METHOD M_GetAllProps : ERRORID
VAR_INPUT
	refCmdData : REFERENCE TO  ST_CmdData;
END_VAR
SUPER^.M_GetAllProps(refCmdData);
nCurrentPropIndex := nCurrentPropIndex + 1;
refCmdData.n32Data[nCurrentPropIndex] := REAL_TO_DINT(rWorkingDistance);
nCurrentPropIndex := nCurrentPropIndex + 1;
refCmdData.n32Data[nCurrentPropIndex] := BOOL_TO_DINT(bInvertWorkingDistance);
nCurrentPropIndex := nCurrentPropIndex + 1;
refCmdData.n32Data[nCurrentPropIndex] := eLightOutput;
nCurrentPropIndex := nCurrentPropIndex + 1;
refCmdData.n32Data[nCurrentPropIndex] := nLightOutputChannel;
END_METHOD

METHOD M_SetAllProps : ERRORID
VAR_INPUT
	refCmdData : REFERENCE TO  ST_CmdData;
END_VAR
M_SetAllProps := SUPER^.M_SetAllProps(refCmdData);

IF M_SetAllProps > 0 THEN
	RETURN;
END_IF

//WorkingDistance
nCurrentPropIndex := nCurrentPropIndex + 1;
nSpecPropIndex := nCurrentPropIndex;
rWorkingDistance := DINT_TO_REAL(refCmdData.n32Data[nCurrentPropIndex]);
nCurrentPropIndex := nCurrentPropIndex + 1;
bInvertWorkingDistance := DINT_TO_BOOL(refCmdData.n32Data[nCurrentPropIndex]);

//LightOutput
nCurrentPropIndex := nCurrentPropIndex + 1;
eLightOutput := DINT_TO_USINT(refCmdData.n32Data[nCurrentPropIndex]);

//LightOutputChannel
nCurrentPropIndex := nCurrentPropIndex + 1;
nLightOutputChannel := DINT_TO_USINT(refCmdData.n32Data[nCurrentPropIndex]);

nNoOfProps := nCurrentPropIndex + 1;
END_METHOD

METHOD M_SetSingleProp : ERRORID
VAR_INPUT
	refCmdData : REFERENCE TO  ST_CmdData;
END_VAR
IF nSpecPropIndex = refCmdData.aHeader[1] THEN
	rWorkingDistance := DINT_TO_REAL(refCmdData.n32Data[0]);
ELSIF nSpecPropIndex + 1 = refCmdData.aHeader[1] THEN
	bInvertWorkingDistance := DINT_TO_BOOL(refCmdData.n32Data[0]);
ELSIF nSpecPropIndex + 3 = refCmdData.aHeader[1] THEN
	nLightOutputChannel := DINT_TO_USINT(refCmdData.n32Data[0]);
ELSE
	M_SetSingleProp := SUPER^.M_SetSingleProp(refCmdData);
END_IF
END_METHOD

PROPERTY P_stAbsPosTotal : ST_3DPoint
GET
VAR
	stPosTemp : ST_3DPoint;
END_VAR
stPosTemp := SUPER^.P_stAbsPosPhys;
IF bInvertWorkingDistance THEN
	stPosTemp.Z := stPosTemp.Z + rWorkingDistance;
ELSE
	stPosTemp.Z := stPosTemp.Z - rWorkingDistance;
END_IF
P_stAbsPosTotal := stPosTemp;
END_GET
END_PROPERTY

PROPERTY P_stCurrentPosTotal : ST_3DPoint
GET
VAR
	stPosTemp : ST_3DPoint;
END_VAR
stPosTemp := P_stCurrentPosPhys;
IF bInvertWorkingDistance THEN
	stPosTemp.Z := stPosTemp.Z + rWorkingDistance;
ELSE
	stPosTemp.Z := stPosTemp.Z - rWorkingDistance;
END_IF
P_stCurrentPosTotal := stPosTemp;
END_GET
END_PROPERTY

END_FUNCTION_BLOCK

// ---- Objects/Tools/FB_ZLevelSensor.TcPOU
FUNCTION_BLOCK FB_ZLevelSensor EXTENDS FB_MzTool
VAR_INPUT
END_VAR
VAR_OUTPUT
END_VAR
VAR
	rCurrentZMeasPos	: REAL;
	rZMeasPosOffset		: REAL;
END_VAR

SUPER^();	//FB_MzTool aufrufen

//Prozessdaten aktualisieren
IF pZAxisRef > 0 THEN
	stProcessData.n32Data[7] := BOOL_TO_DINT(pZAxisRef^.stInput.nToolState.1);
END_IF
aObjProcData[nNotifyId] := stProcessData;

ACTION A_Reset:
nStateA_ResetSpec := 80;
SUPER^.A_Reset();
END_ACTION

METHOD FB_init : BOOL
VAR_INPUT
	bInitRetains : BOOL; // if TRUE, the retain variables are initialized (warm start / cold start)
	bInCopyCode : BOOL;  // if TRUE, the instance afterwards gets moved into the copy code (online change)
END_VAR
eObjectType := E_ObjectType.OBJECTTYPE_ZSensor;
eObjectGroup := E_ObjectGroup.OBJECTGROUP_MzTool OR E_ObjectGroup.OBJECTGROUP_Device;
END_METHOD

METHOD M_AddChild : ERRORID
VAR_INPUT
	pObject : POINTER TO FB_Object;
	nSlotNr	: UINT;
	nIndex 	: INT;
END_VAR
//Kann keine Objekte aufnehmen
M_AddChild := E_ErrorIdObjMgmt.ERRORID_ObjectCanNotTakeChilds;
END_METHOD

METHOD M_CheckAction : ERRORID
VAR_INPUT
	refActionData 	: REFERENCE TO ST_ActionData;
	pCorrelObject	: POINTER TO FB_Object;
END_VAR

VAR
	eMeasureMode : E_MeasureMode;
	pInkStation	 : POINTER TO FB_InkStation;
END_VAR
CASE refActionData.eAction OF
	E_Action.ACTION_MeasureTool:
		//ZSensor montiert?
		IF NOT P_bSensorMounted THEN
			M_CheckAction := E_ErrorIdCmd.ERRORID_ZSensorNotMounted;
		END_IF
		//MeasureMode auswerten
		eMeasureMode := DINT_TO_USINT(refActionData.aParams[1]);
		IF eMeasureMode = E_MeasureMode.MEAS_MODE_Auto THEN	//Target muss passend sein
			CASE fbObjectDirectory.M_GetObjType(refActionData.nTarget) OF
				E_ObjectType.OBJECTTYPE_InkStation:
					pInkStation := fbObjectDirectory.M_GetObjPointer(refActionData.nTarget);
					//Inkstation offen?
					IF (pInkStation^.P_eCoverState <> E_OpClState.Open) THEN
						M_CheckAction := E_ErrorIdCmd.ERRORID_InkStationNotOpen;
						RETURN;
					END_IF
					//Inkstation im Stillstand?
					IF(pInkStation^.P_nCurrentSpinSpeed <> 0) THEN
						M_CheckAction := E_ErrorIdCmd.ERRORID_InkStationIsStillSpinning;
						RETURN;
					END_IF
				E_ObjectType.OBJECTTYPE_DryPad,
				E_ObjectType.OBJECTTYPE_Slide,
				//E_ObjectType.OBJECTTYPE_Wafer,
				E_ObjectType.OBJECTTYPE_Point:
				//Do nothing
			ELSE
				M_CheckAction := E_ErrorIdCmd.ERRORID_UnsuitableTarget;
				RETURN;
			END_CASE
		
		ELSIF eMeasureMode = E_MeasureMode.MEAS_MODE_SemiAuto THEN	//Target muss erst ermittelt werden
			//nMeasToolTargetIdx := aI_MzTool[nMeasToolMzToolIdx].M_GetCurrentTargetIdx();
			//passendes Target gefunden?
			(*IF NOT (aI_Target[nMeasToolTargetIdx].P_eObjectType = E_ObjectType.OBJECTTYPE_Slide OR 
				aI_Target[nMeasToolTargetIdx].P_eObjectType = E_ObjectType.OBJECTTYPE_DryPad OR
				aI_Target[nMeasToolTargetIdx].P_eObjectType = E_ObjectType.OBJECTTYPE_Wafer) THEN
				M_ExeAction := E_ErrorIdCmd.ERRORID_InvalidTarget;
				RETURN;					
			END_IF*)
			;
		ELSE
			M_CheckAction := E_ErrorIdCmd.ERRORID_InvalidMeasureMode;
			RETURN;
		END_IF	
ELSE
	M_CheckAction := SUPER^.M_CheckAction(refActionData, pCorrelObject);	
END_CASE
END_METHOD

METHOD M_SetAllProps : ERRORID
VAR_INPUT
	refCmdData : REFERENCE TO  ST_CmdData;
END_VAR

VAR
	pExtruder : POINTER TO FB_Extruder;
END_VAR
IF pParentMzTool^.P_eObjectType = E_ObjectType.OBJECTTYPE_SinglePiezoHolder THEN
	;	
ELSIF pParentMzTool^.P_eObjectType = E_ObjectType.OBJECTTYPE_Extruder THEN
	pExtruder := pParentMzTool;
	IF pExtruder^.P_eExtruderType <> E_ExtruderType.SyringeExtruder1 THEN
		M_SetAllProps := E_ErrorIdObjMgmt.ERRORID_InvalidParentMzTool;
		RETURN;	
	END_IF
ELSE
	M_SetAllProps := E_ErrorIdObjMgmt.ERRORID_InvalidParentMzTool;
	RETURN;	
END_IF

M_SetAllProps := SUPER^.M_SetAllProps(refCmdData);
END_METHOD

PROPERTY P_bCollFree : BOOL
GET
VAR
	st3DPoint 		: ST_3DPoint;
END_VAR
//wenn Z-Stift nicht montiert, dann kollisionsfrei
IF pZAxisRef^.stInput.nToolState.1 THEN
	P_bCollFree := SUPER^.P_bCollFree;
ELSE
	P_bCollFree := TRUE;
END_IF
END_GET
END_PROPERTY

PROPERTY P_bSensorMounted : BOOL
GET
IF pParentMzTool^.P_eObjectType = E_ObjectType.OBJECTTYPE_SinglePiezoHolder OR pParentMzTool^.P_eObjectType = E_ObjectType.OBJECTTYPE_Extruder THEN
	P_bSensorMounted := pZAxisRef^.stInput.nToolState.1;	
END_IF
END_GET
END_PROPERTY

PROPERTY P_rToolRadius : REAL
GET
VAR
	stDim : ST_3DDimension;
END_VAR
P_rToolRadius := 1500.0;
END_GET
END_PROPERTY

END_FUNCTION_BLOCK

// ---- Objects/Targets/Active/FB_InkStation.TcPOU
FUNCTION_BLOCK FB_InkStation EXTENDS FB_ActiveTarget IMPLEMENTS I_TargetZSensor

VAR
	//Hardware-Verküpfung
	pSpinDrive			: POINTER TO FB_HwRefInkStatDriveSpin;
	pCoverDrive			: POINTER TO FB_HwRefInkStatDriveCover;
	//Hardware-Bausteine
	fbInitSpinDrive		: FB_InkStationInitSpinDrive;
	fbInitSpinCover		: FB_InkStationInitCoverDrive;
	fbOpenCloseCover	: FB_InkStationOpenClose;
	
	
	//Variablen allgemeine Statemachine
	eBasicAction		: E_Action;
	
	//Prozessdaten
	nCurrentSpinSpeed	: INT;
	bVacuumOn			: BOOL;
	
	//Spec-Properties
	nNoOfSpecPoints : USINT;
	stMeasurePoint		: ST_3DPoint;
	stInkPoint			: ST_3DPoint;
	nValveNrVac			: USINT;	//VentilNr Vakuum (FBox)
	nMinHoldVac			: INT;		//minimales Haltevakuum um zu Schleudern
	
	//****************************************Aktionvariablen****************************************************
	bActionLock			: ARRAY[50..150] OF BOOL;
	
	
	//Action: "Spin"
	bSpin				: BOOL;	
	nStateA_Spin		: USINT;			//State von A_Spin();
	
	timerSpin			: TON;				//Timer für Schleuderzeit
	tSpinTime			: TIME; 			//Schleuderzeit (bei 0 wird dauerhaft eingeschalten bis zum Ausschalten)
	nSpinSpeed			: INT;				//Drehzahl Schleuder RPM
	
	//Action: "OpenClose"
	bOpenClose			: BOOL;
	nStateA_OpenClose	: USINT;	//Statemachine von A_OpenClose();
	eOpClCtrl			: E_OpClCtrl;

END_VAR

{IF defined (variable:aFbInkStatDrvSpinRef)}
IF bInitFB THEN
	bInitFB := FALSE;
	F_CreateLinkedListHnd( ADR( aNodes ), SIZEOF( aNodes ), hList );
	//Fehlerstruktur vorausfüllen
	stError.ObjectId := nObjectID;
	stError.HardwareGrp := E_HardwareGrp.Nothing;
	stError.POU := E_POU.POU_FB_InkStation;
END_IF
IF (pSpinDrive = 0) OR  (pCoverDrive = 0) THEN
	RETURN;
END_IF

bIsInit := pSpinDrive^.bIsInit AND pCoverDrive^.bIsInit;
nCurrentSpinSpeed := pSpinDrive^.nCurrentSpeed  * 3;	//RPM

CASE eCurrentState OF
	E_MachineState.MACHINESTATE_Active:
		//BasicActions ausführen
		IF bInit THEN	//Initialisieren
			A_Init();
			IF nStateA_Init >= 80 THEN
				IF nStateA_Init >= 99 THEN
					bError := TRUE;	
				END_IF
				bInit := FALSE;
				nStateA_Init := 0;
				M_RemoveListEntry(nSearchValue:= E_Action.ACTION_Init);
			END_IF
		END_IF
		
		IF bSpin THEN	//Drehzahl Schleuder vorgeben
			A_Spin();
			IF nStateA_Spin >= 80 THEN
				IF nStateA_Spin >= 99 THEN
					bError := TRUE;	
				END_IF
				bSpin := FALSE;
				nStateA_Spin := 0;
				M_RemoveListEntry(nSearchValue:= E_Action.ACTION_InkSpin);
			END_IF
		END_IF		
		
		IF bOpenClose THEN	//Deckel auf/zu
			A_OpenClose();
			IF nStateA_OpenClose >= 80 THEN
				IF nStateA_OpenClose >= 99 THEN
					bError := TRUE;	
				END_IF
				bOpenClose := FALSE;
				nStateA_OpenClose := 0;
				M_RemoveListEntry(nSearchValue:= E_Action.ACTION_InkOpClCover);
			END_IF
		END_IF		
		
		IF bStop THEN
			A_Stop();
			IF nStateA_Stop >= 80 THEN
				IF nStateA_Stop >= 99 THEN
					bError := TRUE;
				END_IF
				M_RemoveListEntry(nSearchValue:= E_Action.ACTION_Stop);
				nStateA_Stop := 0;
				bStop := FALSE;
			END_IF							
		END_IF		
		
		IF hList.nCount = 0 THEN
			eCurrentState := E_MachineState.MACHINESTATE_Ready;
		END_IF

		IF bError  THEN
			eCurrentState := E_MachineState.MACHINESTATE_Error;
		END_IF

	E_MachineState.MACHINESTATE_Reset:
		A_Reset();
		IF nStateA_Reset = 80 THEN
			nStateA_Init := 0;
			nStateA_Spin := 0;
			nStateA_OpenClose := 0;
			nStateA_Stop := 0;
			nStateA_Reset := 0;
			bBusy := FALSE;
			bError := FALSE;
			bStopAllOnError := FALSE;
			fbList.A_Reset( hList := hList);
			MEMSET(ADR(bActionLock),0,SIZEOF(bActionLock));
			nErrorId := 0;
			stError.Cmd := 0;
			stError.ErrorId := 0;
			eCurrentState := E_MachineState.MACHINESTATE_Idle;
		ELSIF
			nStateA_Reset = 99 THEN
			fbErrorList.M_Add(stError);
			nStateA_Reset := 0;
			bBusy := FALSE;
			bError := TRUE;
			eCurrentState := E_MachineState.MACHINESTATE_Error;			
		END_IF
	
	E_MachineState.MACHINESTATE_Ready:
		bBusy := FALSE;
		eCurrentState := E_MachineState.MACHINESTATE_Idle;
	
	E_MachineState.MACHINESTATE_Error:
		pSpinDrive^.nSpeed := 0;
		bBusy := FALSE;
END_CASE

//Prozessdaten aktualisieren
stProcessData.nObjId := nObjectID;
stProcessData.n32Data[0] := BOOL_TO_DINT(bIsInit);
stProcessData.n32Data[1] := eCurrentState;
stProcessData.n32Data[2] := stError.ErrorId;
stProcessData.n32Data[3] := pSpinDrive^.nCurrentSpeed;
stProcessData.n32Data[4] := pCoverDrive^.P_eCoverState;
stProcessData.n32Data[5] := BOOL_TO_DINT(bVacuumOn);
stProcessData.n32Data[6] := pSpinDrive^.nCurrentVacuum;

aObjProcData[nNotifyId] := stProcessData;
{END_IF}

ACTION A_Init:
stError.POUState := nStateA_Init;

CASE nStateA_Init OF
	0:	//Spin initialisieren
		fbInitSpinDrive(pDriveRef:= pSpinDrive, bExecute:= TRUE);
		IF NOT fbInitSpinDrive.bBusy THEN
			IF fbInitSpinDrive.bError THEN
				stError.ErrorId := fbInitSpinDrive.nErrorId;
				nStateA_Init := 99;
			ELSE
				nStateA_Init := 1;			
			END_IF
			fbInitSpinDrive(bExecute:= FALSE);
		END_IF
	
	1: //Cover initialisieren
		fbInitSpinCover(pDriveRef:= pCoverDrive, bExecute:= TRUE);
		IF NOT fbInitSpinCover.bBusy THEN
			IF fbInitSpinCover.bError THEN
				stError.ErrorId := fbInitSpinCover.nErrorId;
				nStateA_Init := 99;
			ELSE
				nStateA_Init := 80;
			END_IF
			fbInitSpinCover(bExecute:= FALSE);
		END_IF
		
	70:	//Abbrechen
		nStateA_Init := 80;
		fbInitSpinDrive();
		IF fbInitSpinDrive.bBusy THEN
			nStateA_Init := 70;
			fbInitSpinDrive.M_Stop();
		ELSE
			fbInitSpinDrive(bExecute:= FALSE);
		END_IF
		fbInitSpinCover();
		IF fbInitSpinCover.bBusy THEN
			nStateA_Init := 70;
			fbInitSpinCover.M_Stop();
		ELSE
			fbInitSpinCover(bExecute:= FALSE);
		END_IF
END_CASE

//Errorhandling
IF nStateA_Init = 99 THEN
	stError.Cmd := E_Action.ACTION_Init;
	stError.POUAction := E_POUACT.POUACT_A_Init;
	fbErrorList.M_Add(stError);
END_IF
END_ACTION

ACTION A_OpenClose:
stError.POUState := nStateA_OpenClose;

IF nStateA_OpenClose = 0 THEN
	fbOpenCloseCover(pDriveRef:= pCoverDrive, eCtrl:= eOpClCtrl, bExecute:= TRUE); 
	IF NOT fbOpenCloseCover.bBusy THEN
		IF fbOpenCloseCover.bError THEN
			stError.ErrorId := fbOpenCloseCover.nErrorId;
			nStateA_OpenClose := 99;
		ELSE
			nStateA_OpenClose := 80;
		END_IF
		fbOpenCloseCover(bExecute:= FALSE); 
	END_IF
END_IF

//Errorhandling
IF nStateA_OpenClose = 99 THEN
	stError.Cmd := E_Action.ACTION_InkOpClCover;
	stError.POUAction := E_POUACT.POUACT_A_OpenClose;
	fbErrorList.M_Add(stError);
END_IF
END_ACTION

ACTION A_Reset:
CASE nStateA_Reset OF
	0:
		nStateA_Reset := 80;
END_CASE
END_ACTION

ACTION A_Spin:
IF pSpinDrive^.nStatus.3 THEN	//Error
	stError.POUState := nStateA_Spin;
	nStateA_Spin := 99;
END_IF

CASE nStateA_Spin OF
	0:
		pSpinDrive^.nSpeed := nSpinSpeed;
		IF tSpinTime > T#0S THEN
			timerSpin(IN:= TRUE, PT:= tSpinTime);
		END_IF
		nStateA_Spin := 1;
		
	1:	//Überwachung Vacuum, Timer, Drezahl
		pSpinDrive^.nSpeed := nSpinSpeed;
		timerSpin();
		IF timerSpin.Q OR (pSpinDrive^.nSpeed = 0 AND pSpinDrive^.nCurrentSpeed = 0) OR nMinHoldVac < pSpinDrive^.nCurrentVacuum THEN
			timerSpin(IN:= FALSE);	
			pSpinDrive^.nSpeed := 0;
			nStateA_Spin := 2;
		END_IF
		
	2:	//Warten bis Drehzahl auf 0
		IF pSpinDrive^.nCurrentSpeed = 0 THEN
			nStateA_Spin := 80;
		END_IF
		
	70:	//Abbrechen
		timerSpin(IN:= FALSE);
		pSpinDrive^.nSpeed := 0;
		nStateA_Spin := 71;
		
	71:	//Speed = 0?
		IF pSpinDrive^.nCurrentSpeed = 0 THEN
			nStateA_Spin := 80;
		END_IF
		
END_CASE

//Errorhandling
IF nStateA_Spin = 99 THEN
	stError.Cmd := E_Action.ACTION_InkSpin;
	stError.POUAction := E_POUACT.POUACT_A_Spin;
	fbErrorList.M_Add(stError);
END_IF
END_ACTION

ACTION A_Stop:
CASE nStateA_Stop OF
	0:	
		IF bInit THEN
			nStateA_Init := 70;	
		END_IF
		
		IF bSpin THEN
			nStateA_Spin := 70;
		END_IF
		
		nStateA_Stop := 1;
	
	1:	//Warten bis alle Actions außer Stop abgebrochen sind
		IF hList.nCount = 1 THEN	//nur der Eintrag von Stop
			nStateA_Stop := 80;
		END_IF
END_CASE

//Errorhandling
IF nStateA_Stop = 99 THEN
	stError.Cmd := E_Action.ACTION_Stop;
	stError.POUAction := E_POUACT.POUACT_A_Stop;
	fbErrorList.M_Add(stError);
END_IF
END_ACTION

METHOD FB_init : BOOL
VAR_INPUT
	bInitRetains : BOOL; // if TRUE, the retain variables are initialized (warm start / cold start)
	bInCopyCode : BOOL;  // if TRUE, the instance afterwards gets moved into the copy code (online change)
END_VAR
eObjectType := E_ObjectType.OBJECTTYPE_InkStation;
eObjectGroup := E_ObjectGroup.OBJECTGROUP_Target OR E_ObjectGroup.OBJECTGROUP_Device;
END_METHOD

METHOD M_ApplyPos : ERRORID
VAR_INPUT
	eTargetRef 		: E_TargetRef;
	nPointSlotNr	: UINT;
	stPos 			: ST_3DPoint;
	bXPos			: BOOL;
	bYPos			: BOOL;
	bZPos			: BOOL;	
END_VAR
VAR
	stAbsPos		: ST_3DPoint;
END_VAR
IF eTargetRef = E_TargetRef.TARGETREF_SpecPoint THEN
	IF nPointSlotNr = 2 THEN
		stAbsPos := P_stAbsPosLB;
		IF bXPos THEN
			stInkPoint.X := stPos.X - stAbsPos.X;
		END_IF
		IF bYPos THEN
			stInkPoint.Y := stPos.Y - stAbsPos.Y;
		END_IF
		IF bZPos THEN
			stInkPoint.Z := stPos.Z - stAbsPos.Z;
		END_IF
	ELSE
		M_ApplyPos := E_ErrorIdCmd.ERRORID_InvalidTargetPointNr;
	END_IF
ELSE
	M_ApplyPos := SUPER^.M_ApplyPos(eTargetRef, nPointSlotNr, stPos, bXPos, bYPos, bZPos);
END_IF
END_METHOD

METHOD M_CancelAction
VAR_INPUT
	eAction : E_Action;
END_VAR
IF eAction = E_Action.ACTION_InkSpin THEN
	M_Stop();
END_IF
END_METHOD

METHOD M_CheckAction : ERRORID
VAR_INPUT
	refActionData 	: REFERENCE TO ST_ActionData;
	pCorrelObject	: POINTER TO FB_Object;
END_VAR
IF refActionData.eAction = E_Action.ACTION_TeachTarget THEN
	IF NOT DINT_TO_UINT(refActionData.aParams[1]) = E_TargetRef.TARGETREF_SpecPoint AND refActionData.aParams[2] = 2 THEN
		M_CheckAction := E_ErrorIdCmd.ERRORID_InvalidTargetPointRef;
	END_IF
ELSIF refActionData.eAction = E_Action.ACTION_MoveToTarget THEN
	//Target = Inkpoint -> Inkstation muss geöffnet sein
	IF (refActionData.aParams[1] = E_TargetRef.TARGETREF_SpecPoint) AND (refActionData.aParams[2] = 2) THEN
		IF P_eCoverState <> E_OpClState.Open THEN
			M_CheckAction := E_ErrorIdCmd.ERRORID_InkStationNotOpen;
			RETURN;
		END_IF
		IF P_nCurrentSpinSpeed <> 0 THEN
			M_CheckAction := E_ErrorIdCmd.ERRORID_InkStationIsStillSpinning; //Error
			RETURN;		
		END_IF		
	END_IF
END_IF
END_METHOD

METHOD M_ExeAction : ERRORID
VAR_INPUT
	refActionData	: REFERENCE TO ST_ActionData;	
END_VAR
CASE refActionData.eAction OF
	E_Action.ACTION_Init:
		IF NOT bInit THEN
			bInit := TRUE;
			fbList.A_AddHeadValue(hList := hList, putValue:= E_Action.ACTION_Init);
		ELSE
			RETURN;
		END_IF
		
	E_Action.ACTION_InkSpin:
		nSpinSpeed := DINT_TO_INT(refActionData.aParams[2]);
		nSpinSpeed := nSpinSpeed / 3;		//Velo umrechnen (Übersetzung 1:3)
		tSpinTime := DINT_TO_TIME(refActionData.aParams[3]);
		
		IF NOT bSpin THEN
			IF refActionData.aParams[1] = 1 AND nSpinSpeed <> 0 THEN
				IF nSpinSpeed <> 0 THEN
					IF nMinHoldVac < pSpinDrive^.nCurrentVacuum THEN
						M_ExeAction := E_ErrorIdCmd.ERRORID_VacuumNotOk;  //Error
						RETURN;
					END_IF
				END_IF
			END_IF
		ELSE
			IF refActionData.aParams[1] = 0 THEN
				nSpinSpeed := 0;
			END_IF
		END_IF
		
		getPosPtr := 0;	//nach vorhandenem Eintrag suchen - beginnen an Anfang
		fbList.A_FindNext(hList := hList, putPosPtr := getPosPtr, putValue := E_Action.ACTION_InkSpin, getValue=>getValue, getPosPtr=>getPosPtr );
		IF NOT fbList.bOk THEN	//Eintrag wurde nicht gefunden
			bSpin := TRUE;
			fbList.A_AddHeadValue(hList := hList, putValue:= E_Action.ACTION_InkSpin);
		ELSE
			RETURN;
		END_IF

	E_Action.ACTION_InkOpClCover:
		IF NOT bOpenClose THEN
			IF NOT P_bCoverAreaIsFree THEN
				M_ExeAction := E_ErrorIdCmd.ERRORID_InkStatCoverAreaNotFree;  //Error
				RETURN;
			END_IF
			eOpClCtrl := DINT_TO_USINT(refActionData.aParams[1]);
			fbList.A_AddHeadValue(hList := hList, putValue:= E_Action.ACTION_InkOpClCover);
			bOpenClose := TRUE;
		ELSE
			RETURN;
		END_IF
		
	E_Action.ACTION_SwitchPressure:
		IF refActionData.aParams[1] = 0 THEN
			aValves[nValveNrVac].M_Off();
			bVacuumOn := FALSE;
		ELSE
			aValves[nValveNrVac].M_On(1);
			bVacuumOn := TRUE;
		END_IF
	
	E_Action.ACTION_Stop:
		IF hList.nCount > 0 THEN
			fbList.A_AddHeadValue(hList := hList, putValue:= E_Action.ACTION_Stop);
		ELSE
			RETURN;	
		END_IF
	ELSE
		M_ExeAction := E_ErrorIdCmd.ERRORID_InvalidAction;
END_CASE

eCurrentState := E_MachineState.MACHINESTATE_Active;
bBusy := TRUE;
END_METHOD

METHOD M_GetAbsPos : ST_3DPoint
VAR_INPUT
	pChildPos	: POINTER TO ST_3DPoint;
	eTargetRef 	: E_TargetRef;
	nParam1		: UINT;
 	nParam2		: UINT;
	nParam3		: USINT;
	nParam4		: USINT;
	nZLevel		: USINT;
END_VAR
VAR_OUTPUT
	nErrorId 	: ERRORID;
	lrAngle		: LREAL;
END_VAR
VAR
	stLocPosLB : ST_3DPoint;
END_VAR
IF eTargetRef = E_TargetRef.TARGETREF_SpecPoint THEN
	stLocPosLB := P_stRelPosLB;
	IF nParam1 = 1 THEN	//MeasurePoint
		stLocPosLB := F_Add3DPoints(stLocPosLB,stMeasurePoint);
	ELSIF nParam1 = 2 THEN	//InkPoint
		stLocPosLB := F_Add3DPoints(stLocPosLB,stInkPoint);
	ELSE
		nErrorId := E_ErrorIdCmd.ERRORID_InvalidTargetPointNr;
		RETURN;
	END_IF
	M_GetAbsPos := pParentTarget^.M_GetAbsPos(pChildPos := ADR(stLocPosLB), eTargetRef:= E_TargetRef.TARGETREF_LeftBottom,
												nParam1:= 0,
												nParam2:= 0, nParam3:= 0,nParam4:= 0, nZLevel:= 0,
												lrAngle => lrAngle, nErrorId=> nErrorId);	
ELSE
	M_GetAbsPos := SUPER^.M_GetAbsPos(pChildPos := pChildPos, eTargetRef:= eTargetRef,
													nParam1:= nParam1,
													nParam2:= nParam2, nParam3:= nParam3, nParam4:= 0, nZLevel:= nZLevel,
													lrAngle => lrAngle, nErrorId=> nErrorId);		
END_IF
END_METHOD

METHOD M_GetActionBusy : BOOL
VAR_INPUT
	eAction : E_Action;
END_VAR
getPosPtr := 0;(* start from first node element *)
fbList.A_FindNext( hList := hList, putPosPtr := getPosPtr, putValue := eAction, getValue=>getValue, getPosPtr=>getPosPtr );
IF fbList.bOk THEN	//Eintrag wurde gefunden, d.h. Action ist noch busy
	M_GetActionBusy := TRUE;
END_IF
END_METHOD

METHOD M_GetAllProps : ERRORID
VAR_INPUT
	refCmdData : REFERENCE TO  ST_CmdData;
END_VAR
SUPER^.M_GetAllProps(refCmdData);

nCurrentPropIndex := nCurrentPropIndex + 1;
refCmdData.n32Data[nCurrentPropIndex] := nNoOfSpecPoints;
nCurrentPropIndex := nCurrentPropIndex + 1;
refCmdData.n32Data[nCurrentPropIndex] := REAL_TO_DINT(stMeasurePoint.X);
nCurrentPropIndex := nCurrentPropIndex + 1; 	
refCmdData.n32Data[nCurrentPropIndex] := REAL_TO_DINT(stMeasurePoint.Y);
nCurrentPropIndex := nCurrentPropIndex + 1;
refCmdData.n32Data[nCurrentPropIndex] := REAL_TO_DINT(stMeasurePoint.Z);
nCurrentPropIndex := nCurrentPropIndex + 1;
refCmdData.n32Data[nCurrentPropIndex] := REAL_TO_DINT(stInkPoint.X);
nCurrentPropIndex := nCurrentPropIndex + 1;
refCmdData.n32Data[nCurrentPropIndex] := REAL_TO_DINT(stInkPoint.Y);
nCurrentPropIndex := nCurrentPropIndex + 1;
refCmdData.n32Data[nCurrentPropIndex] := REAL_TO_DINT(stInkPoint.Z);
nCurrentPropIndex := nCurrentPropIndex + 1;
refCmdData.n32Data[nCurrentPropIndex] := REAL_TO_DINT(rZOffset);
nCurrentPropIndex := nCurrentPropIndex + 1;
refCmdData.n32Data[nCurrentPropIndex] := nValveNrVac;
nCurrentPropIndex := nCurrentPropIndex + 1;
refCmdData.n32Data[nCurrentPropIndex] := nMinHoldVac;
END_METHOD

METHOD M_GetProcData : DINT
VAR_INPUT
	eProcDataType : E_ProcDataType;
END_VAR
END_METHOD

METHOD M_RemoveListEntry : BOOL
VAR_INPUT
	nSearchValue	: E_Action;
END_VAR
getPosPtr := 0;(* start from first node element *)
fbList.A_FindNext( hList := hList, putPosPtr := getPosPtr, putValue := nSearchValue, getValue=>getValue, getPosPtr=>getPosPtr );
IF fbList.bOk THEN	//Eintrag wurde gefunden
	fbList.A_RemoveValueAtPosPtr(hList:= hList,	putPosPtr:= getPosPtr);
	IF fbList.bOk THEN
		M_RemoveListEntry := TRUE;
	END_IF
END_IF
END_METHOD

METHOD M_SetAllProps : ERRORID
VAR_INPUT
	refCmdData : REFERENCE TO  ST_CmdData;
END_VAR
{IF defined (variable:aFbInkStatDrvSpinRef)}
pSpinDrive := ADR(aFbInkStatDrvSpinRef[1]);
{ELSE}
{warning 'implement errorId}
M_SetAllProps := 5555;
{END_IF}

{IF defined (variable:aFbInkStatDrvSpinRef)}
pCoverDrive := ADR(aFbInkStatDrvCoverRef[1]);
{ELSE}
{warning 'implement errorId}
M_SetAllProps := 5555;
{END_IF}

M_SetAllProps := SUPER^.M_SetAllProps(refCmdData);

IF M_SetAllProps > 0 THEN
	RETURN;
END_IF

nCurrentPropIndex := nCurrentPropIndex + 1;
nSpecPropIndex := nCurrentPropIndex;
nNoOfSpecPoints := DINT_TO_USINT(refCmdData.n32Data[nCurrentPropIndex]);
nCurrentPropIndex := nCurrentPropIndex + 1;
stMeasurePoint.X := DINT_TO_REAL(refCmdData.n32Data[nCurrentPropIndex]);
nCurrentPropIndex := nCurrentPropIndex + 1;
stMeasurePoint.Y := DINT_TO_REAL(refCmdData.n32Data[nCurrentPropIndex]);
nCurrentPropIndex := nCurrentPropIndex + 1;
stMeasurePoint.Z := DINT_TO_REAL(refCmdData.n32Data[nCurrentPropIndex]);
nCurrentPropIndex := nCurrentPropIndex + 1;
stInkPoint.X := DINT_TO_REAL(refCmdData.n32Data[nCurrentPropIndex]);
nCurrentPropIndex := nCurrentPropIndex + 1;
stInkPoint.Y := DINT_TO_REAL(refCmdData.n32Data[nCurrentPropIndex]);
nCurrentPropIndex := nCurrentPropIndex + 1;
stInkPoint.Z := DINT_TO_REAL(refCmdData.n32Data[nCurrentPropIndex]);
nCurrentPropIndex := nCurrentPropIndex + 1;
rZOffset := DINT_TO_REAL(refCmdData.n32Data[nCurrentPropIndex]);
nCurrentPropIndex := nCurrentPropIndex + 1;
IF refCmdData.n32Data[nCurrentPropIndex] > 0 AND refCmdData.n32Data[nCurrentPropIndex] <= cNoOfValves THEN
	nValveNrVac := DINT_TO_USINT(refCmdData.n32Data[nCurrentPropIndex]);
ELSE
	M_SetAllProps := E_ErrorIdObjMgmt.ERRORID_InvalidValveNumber;
	RETURN;
END_IF
nCurrentPropIndex := nCurrentPropIndex + 1;
nMinHoldVac := DINT_TO_INT(refCmdData.n32Data[nCurrentPropIndex]);
nNoOfProps := nCurrentPropIndex + 1;
END_METHOD

METHOD M_SetSingleProp : ERRORID
VAR_INPUT
	refCmdData : REFERENCE TO  ST_CmdData;
END_VAR

VAR
	nValve : USINT;
END_VAR
IF nSpecPropIndex = refCmdData.aHeader[1] THEN
	M_SetSingleProp := E_ErrorIdCmd.ERRORID_InvalidProperty; //Anzahl SpecPoints darf nicht verändert werden
ELSIF (nSpecPropIndex + 1) = refCmdData.aHeader[1] THEN
	stMeasurePoint.X := DINT_TO_REAL(refCmdData.n32Data[0]);
ELSIF (nSpecPropIndex + 2) = refCmdData.aHeader[1] THEN
	stMeasurePoint.Y := DINT_TO_REAL(refCmdData.n32Data[0]);
ELSIF (nSpecPropIndex + 3) = refCmdData.aHeader[1] THEN
	stMeasurePoint.Z := DINT_TO_REAL(refCmdData.n32Data[0]);
ELSIF (nSpecPropIndex + 4) = refCmdData.aHeader[1] THEN
	stInkPoint.X := DINT_TO_REAL(refCmdData.n32Data[0]);
ELSIF (nSpecPropIndex + 5) = refCmdData.aHeader[1] THEN
	stInkPoint.Y := DINT_TO_REAL(refCmdData.n32Data[0]);
ELSIF (nSpecPropIndex + 6) = refCmdData.aHeader[1] THEN
	stInkPoint.Z := DINT_TO_REAL(refCmdData.n32Data[0]);
ELSIF (nSpecPropIndex + 7) = refCmdData.aHeader[1] THEN
	rZOffset := DINT_TO_REAL(refCmdData.n32Data[0]);
ELSIF (nSpecPropIndex + 8) = refCmdData.aHeader[1] THEN
		nValve := DINT_TO_USINT(refCmdData.n32Data[0]);
		IF nValve > 0 AND nValve <= cNoOfValves THEN
			nValveNrVac := nValve;
		ELSE
			M_SetSingleProp := E_ErrorIdObjMgmt.ERRORID_InvalidValveNumber;	
		END_IF
	
ELSIF (nSpecPropIndex + 9) = refCmdData.aHeader[1] THEN
	nMinHoldVac := DINT_TO_INT(refCmdData.n32Data[0]);	
ELSE
	M_SetSingleProp := SUPER^.M_SetSingleProp(refCmdData);
END_IF
END_METHOD

PROPERTY P_bCoverAreaIsFree : BOOL
GET
VAR
	i : UINT;
	stCurPosMzTool	: ST_3DPoint;
	stCurPosInkStat	: ST_3DPoint;
END_VAR
//Checken, ob sich im Bewegungsbereich des Deckel ein MzTool befindet
P_bCoverAreaIsFree := TRUE;
//Hier stoße ich wieder genau auf das Problem, dass ich ich alle Tools des Heads durchiterieren muss
//Den Head habe ich zur Verfügung
//der Head könnte eine Property zur Verfügung stellen, die einen Pointer auf die Liste der ChildTools zur Verfügung stellt
//Ein Problem könnte aber darstellen, dass wenn bei rekursivem Aufruf der Liste es zu einem Durcheinander kommt.
//Eine sehr gute Idee wäre der Iteratoransatz
//Eine Liste muss damit immer mit Hilfe eins Iterators iteriert werden.
//Wenn begonnen wird zu iterieren, muss dieser resettet werden.
//Bei TwinCAT Vision abschauen!



(*FOR i:= 1 TO fbObjectDirectory.nCntMzTool BY 1 DO
	IF NOT (aI_MzTool[i].P_eObjectType = E_ObjectType.OBJECTTYPE_MZHead) THEN
		IF NOT aI_MzTool[i].P_bCollFree THEN	//Tool ist nicht im kollisionsfreiem Bereich
			
			stCurPosMzTool := aI_MzTool[i].P_stCurrentPosPhys;
			stCurPosInkStat := P_stAbsPosLB;
			IF (stCurPosMzTool.Z - 5000) < stCurPosInkStat.Z THEN
				IF stCurPosMzTool.X >= stCurPosInkStat.X AND stCurPosMzTool.X <= (stCurPosInkStat.X + stDimension.Width)
				AND stCurPosMzTool.Y >= stCurPosInkStat.Y AND stCurPosMzTool.Y <= (stCurPosInkStat.Y + stDimension.Depth) THEN
					P_bCoverAreaIsFree := FALSE;
					RETURN;
				END_IF
			END_IF
 		END_IF
	END_IF
END_FOR*)
END_GET
END_PROPERTY

PROPERTY P_bIsSpinning : BOOL
GET
IF pSpinDrive > 0 THEN
	IF pSpinDrive^.nCurrentSpeed <> 0 THEN
		P_bIsSpinning := TRUE;
	END_IF	
END_IF
END_GET
END_PROPERTY

PROPERTY P_bSensor : BOOL
GET
IF pSpinDrive > 0 THEN
	P_bSensor := pSpinDrive^.bZSensor;	
END_IF
END_GET
END_PROPERTY

PROPERTY P_eCoverState : E_OpClState
GET
P_eCoverState := pCoverDrive^.P_eCoverState;
END_GET
END_PROPERTY

PROPERTY P_nCurrentSpinSpeed : INT
GET
P_nCurrentSpinSpeed := nCurrentSpinSpeed;
END_GET
END_PROPERTY

END_FUNCTION_BLOCK

// ---- Hardware/InkStation/FB_HwRefInkStatDriveSpin.TcPOU
FUNCTION_BLOCK FB_HwRefInkStatDriveSpin EXTENDS FB_CanNodeBase
VAR_INPUT
	//Ausgänge
	nControl		AT %Q* : UINT; 	//Controlword
	nOpMode			AT %Q* : USINT;	//Mode of Operations
	nSpeed			AT %Q* : INT;	//Speed
	bDigiOut0		AT %Q* : BOOL;	//Digitaler Ausgang0
	bDigiOut1		AT %Q* : BOOL;	//Digitaler Ausgang1
	bIsInit 		: BOOL;
END_VAR
VAR_OUTPUT
	//Eingänge
	nStatus	 		AT %I* : UINT;	//Statusword
	nCurrentOpMode	AT %I* : USINT; //Aktueller Wert von Mode of Operation
	bHallSens		AT %I* : BOOL;	//Hall-Sensor
	bZSensor		AT %I* : BOOL;	//ZSensor
	nCurrentSpeed	AT %I* : INT;	//Aktuelle Drehzahl
	nCurrentVacuum : INT;
END_VAR
VAR
	timer : TON;
	nState	: USINT;
END_VAR

IF bNodeEnabled THEN
	SUPER^();
	//Vacuum abrufen alle 1s
	IF bIsInit THEN
		CASE nState OF
			0:	//Analogwert per SDO auslesen
				fbSdoRead(sADSNetID:= stAdsAdress.sNetId,nPortNr:= stAdsAdress.nPort,
						nIndex:= 16#270E, nSubIndex:= 1, nDataLength:= 4, bExecute:= TRUE);
						
				IF NOT fbSdoRead.bBusy THEN
					IF NOT fbSdoRead.bError THEN
						//Vacuum-Sensor misst den Absolutdruck.
						//Messbereich 20-400kPa (absolut) bei Ausgangsspannung 0,2V - 4,8V
						//als atmosphärischer Druck wird 100kPa angenommen
						nCurrentVacuum := REAL_TO_INT((F_YFuncX(rxMin:= 0.2, rxMax:= 4.8,
												ryMin:= 20.0, ryMax:= 400.0,
												rx:= 10.0/4095.0* DINT_TO_REAL(fbSdoRead.nData))) - 100.0);
						
						fbSdoRead(bExecute:= FALSE);
						
					END_IF
					nState := 1;
				END_IF
				
			1:	//Warten
				timer(IN:= TRUE, PT:= T#1S);
				IF timer.Q THEN
					timer(IN:= FALSE);
					nState := 0;
				END_IF
		END_CASE
		
		//LED-Anzeige (nur bei manchen Bauformen)
		IF nCurrentSpeed = 0 THEN
			bDigiOut0 := FALSE;
		ELSE
			bDigiOut0 := TRUE;
		END_IF
		
	ELSE
		nCurrentVacuum := 0;
 	END_IF
	
END_IF

END_FUNCTION_BLOCK

// ---- Hardware/InkStation/FB_HwRefInkStatDriveCover.TcPOU
FUNCTION_BLOCK FB_HwRefInkStatDriveCover EXTENDS FB_CanNodeBase
VAR_INPUT
	//Ausgänge
	nControl		AT %Q* : UINT; 	//Controlword
	nOpMode			AT %Q* : USINT;	//Mode of Operations
	nTargetPos		AT %Q* : DINT;	//Target Position
	bDigiOut0		AT %Q* : BOOL;	//Digitaler Ausgang0
	bDigiOut1		AT %Q* : BOOL;	//Digitaler Ausgang1
	bIsInit 		: BOOL;
END_VAR
VAR_OUTPUT
	//Eingänge
	nStatus	 		AT %I* : UINT;	//Statusword
	nCurrentOpMode	AT %I* : USINT; //Aktueller Wert von Mode of Operation
	bClosedSwitch	AT %I* : BOOL;	//LimitSwitch Deckel geschlossen
	bOpenSwitch		AT %I* : BOOL;	//LimitSwitch Deckel geöffnet
	
END_VAR
VAR
	eCoverState		: E_OpClState;
END_VAR

IF bNodeEnabled THEN
	SUPER^();	
END_IF

PROPERTY P_eCoverState : E_OpClState
SET
eCoverState := P_eCoverState;
END_SET
GET
P_eCoverState := eCoverState;
END_GET
END_PROPERTY

END_FUNCTION_BLOCK

// ---- Hardware/InkStation/FB_InkStationInitSpinDrive.TcPOU
FUNCTION_BLOCK FB_InkStationInitSpinDrive
VAR_INPUT
	pDriveRef		: POINTER TO FB_HwRefInkStatDriveSpin;
	bExecute		: BOOL;
END_VAR
VAR_OUTPUT
	bBusy		: BOOL;
	bError		: BOOL;
	nErrorId	: ERRORID;
END_VAR
VAR
	fbSdoWrite	: FB_SDO_WRITE;
	fbPower		: FB_CANOpenMotionPower;
	nState		: USINT;
	
	nStateA 		: USINT;
	nStateANext 	: USINT;
	bCancel			: BOOL;
	
	dwSdoIndex 		: DWORD;
	dwSdoSubIndex 	: DWORD;
	dwSdoDataLength : DWORD;
	nSdoDataValue 	: DINT;
	
END_VAR

IF bExecute THEN
	CASE nState OF
		0:	//Prepare
			bBusy := TRUE;
			pDriveRef^.bIsInit := FALSE;
			A_Prepare();
			IF nStateA >= 80 THEN
				IF nStateA >= 99 THEN
					bError := TRUE;
					bBusy := FALSE;
					nState := 99;
				ELSE
					IF bCancel THEN
						nState := 80;
						bBusy := FALSE;
					ELSE
						nState := 1;	
					END_IF
				END_IF
			END_IF

		1:	//PowerOn
			fbPower(pControl:= ADR(pDriveRef^.nControl), pStatus:= ADR(pDriveRef^.nStatus), bExecute:= TRUE);
			IF NOT 	fbPower.bBusy THEN
				IF fbPower.bError THEN
					bError := TRUE;
					bBusy := FALSE;
					nState := 99;
				ELSE
					pDriveRef^.bDigiOut1 := TRUE;	//Versorgung für Digitale IOs (5V) einschalten
					pDriveRef^.nOpMode := 2; 		//Mode = Velocity-Mode
					bBusy := FALSE;
					pDriveRef^.bIsInit := TRUE;
				END_IF
				fbPower(bExecute:= FALSE);
			END_IF
			IF bCancel THEN
				fbPower(bExecute:= FALSE);
				bBusy := FALSE;	
			END_IF
	END_CASE
ELSE
	bError := FALSE;
	bCancel := FALSE;
	nErrorId := 0;
	nState := 0;
END_IF

ACTION A_Prepare:
CASE nStateA OF
	0:	//Errorbit gesetzt?
			IF pDriveRef^.nStatus.3 THEN //Error zurücksetzen
				pDriveRef^.nControl := 153;
			ELSE
				pDriveRef^.nControl := 0;
				nStateA := 1;
			END_IF
			
	1:	//Velocity Dimension Index auf Internal units setzen (sonst lässt sich Microstepping nicht setzen)
		dwSdoIndex := 16#208C;
		dwSdoSubIndex := 0;
		dwSdoDataLength := 1;
		nSdoDataValue := 0; //Internal Units
		nStateANext := 2;
		nStateA := 60; //Sdo senden			
		
	2:	//Microstepping auf 128-fach setzen
		dwSdoIndex := 16#2000;
		dwSdoSubIndex := 0;
		dwSdoDataLength := 1;
		nSdoDataValue := 7; //Microstepping 128-fach
		nStateANext := 3;
		nStateA := 60; //Sdo senden			
			
	3:	//Pulsedivisor auf 0 setzen
		dwSdoIndex := 16#2086;
		dwSdoSubIndex := 0;
		dwSdoDataLength := 1;
		nSdoDataValue := 0; //Pulsedivisor 0
		nStateANext := 4;
		nStateA := 60; //Sdo senden			
			
	4:	//SwitchParameters setzen (keine Endlagen verwenden)		
		dwSdoIndex := 16#2005;
		dwSdoSubIndex := 0;
		dwSdoDataLength := 4;
		nSdoDataValue := 3; //keine Endlagen
		nStateANext := 5;
		nStateA := 60; //Sdo senden			
			
	5:	//Brake deaktivieren			
		dwSdoIndex := 16#200C;
		dwSdoSubIndex := 2;
		dwSdoDataLength := 1;
		nSdoDataValue := 0; //keine Brake
		nStateANext := 6;
		nStateA := 60; //Sdo senden

	6:	//Digital Outputmask setzen		
		dwSdoIndex := 16#2703;
		dwSdoSubIndex := 2;
		dwSdoDataLength := 4;
		nSdoDataValue := 16#30000; //Mask
		nStateANext := 7;
		nStateA := 60; //Sdo senden
		
	7:	//MaxCurrent setzen
		dwSdoIndex := 16#2003;
		dwSdoSubIndex := 0;
		dwSdoDataLength := 1;
		nSdoDataValue := 170; //max Current (max255)
		nStateANext := 8;
		nStateA := 60; //Sdo senden
		
	8:	//Velocity Dimension Index setzen in RPM (Umdrehungen pro min)
		dwSdoIndex := 16#208C;
		dwSdoSubIndex := 0;
		dwSdoDataLength := 1;
		nSdoDataValue := 164; //164 ist Code für RPM
		nStateANext := 9;
		nStateA := 60; //Sdo senden
		
	9:	//vl Velocity Acc DeltaSpeed setzen (Dec wird automatisch gleich gesetzt)
		dwSdoIndex := 16#6048;
		dwSdoSubIndex := 1;
		dwSdoDataLength := 4;
		nSdoDataValue := 100;
		nStateANext := 80;
		nStateA := 60; //Sdo senden		
			
	60:	//Send SDO
		fbSdoWrite(sADSNetID:= pDriveRef^.stAdsAdress.sNetId,nPortNr:= pDriveRef^.stAdsAdress.nPort, 
					nIndex:= dwSdoIndex, nSubIndex:= dwSdoSubIndex, nDataLength:= dwSdoDataLength,
					 nData:= nSdoDataValue, bExecute:= TRUE);
		IF NOT fbSdoWrite.bBusy THEN
			IF fbSdoWrite.bError THEN
				nErrorId := fbSdoWrite.nAdsErrorId;
				nStateA := 99;
			ELSE
				nStateA := nStateANext;
			END_IF
			fbSdoWrite(bExecute:= FALSE);
		END_IF
		
	70:	//Abbrechen
		IF fbSdoWrite.bBusy THEN
			fbSdoWrite(bExecute:= FALSE);
			nStateA := 80;
		END_IF
END_CASE
END_ACTION

METHOD M_Stop
VAR_INPUT
END_VAR
IF bBusy THEN
	bCancel := TRUE;
END_IF
END_METHOD

END_FUNCTION_BLOCK

// ---- Hardware/FB_CANOpenMotionPower.TcPOU
FUNCTION_BLOCK FB_CANOpenMotionPower
VAR_INPUT
	bExecute 	: BOOL;
	pStatus 	: POINTER TO UINT;
	pControl 	: POINTER TO UINT;
END_VAR
VAR_OUTPUT
	bBusy	: BOOL;
	bError	: BOOL;
END_VAR
VAR
	nState : USINT;
END_VAR

IF bExecute THEN
	CASE nState OF
		0:	//Error?
			bBusy := TRUE;
			IF F_GetCoDS402State(pStatus^) = E_CoDS402States.DS402STATE_Fault THEN  //Error
				pControl^ := 153;
			ELSE
				pControl^ := 0;
				nState := 1;
			END_IF
			
		1:	//Leistungsteil einschalten - "Ready to switch on"
			pControl^ := 6;
			nState := 2;
			
		2:	//Abfrage auf Status "Ready to switch on"
			IF F_GetCoDS402State(pStatus^) = E_CoDS402States.DS402STATE_Fault THEN  //Error
				nState := 99;
			ELSIF F_GetCoDS402State(pStatus^) = E_CoDS402States.DS402STATE_ReadyToSwitchOn  THEN//"Ready to switch on"
				nState := 3;
			END_IF
			
		3:	//Leistungsteil einschalten - "Switch on" und "Voltage Enabled"
			pControl^ := 7;
			nState := 4;
			
		4:	//Abfrage auf Status "Switch on" und "Voltage Enabled"
			IF F_GetCoDS402State(pStatus^) = E_CoDS402States.DS402STATE_Fault THEN  //Error
				nState := 99;
			ELSIF F_GetCoDS402State(pStatus^) = E_CoDS402States.DS402STATE_SwitchedOn THEN //"Switch on" und "Voltage Enabled"
				nState := 5;
			END_IF
			
		5:	//Leistungsteil einschalten - "Operation Enabled"
			pControl^ := 15;
			nState := 6;		
	
		6:	//Abfrage auf Status "Operation Enabled"
			IF F_GetCoDS402State(pStatus^) = E_CoDS402States.DS402STATE_Fault THEN  //Error
				nState := 99;
			ELSIF F_GetCoDS402State(pStatus^) = E_CoDS402States.DS402STATE_OperationEnabled THEN //"Operation Enabled"
				bBusy := FALSE;
			END_IF
	END_CASE
	
	IF nState = 99 THEN
		bError := TRUE;
		bBusy := FALSE;
	END_IF
ELSE
	bError := FALSE;
	bBusy := FALSE;
	nState := 0;
END_IF

END_FUNCTION_BLOCK

// ---- Hardware/InkStation/FB_InkStationInitCoverDrive.TcPOU
FUNCTION_BLOCK FB_InkStationInitCoverDrive
VAR_INPUT
	pDriveRef		: POINTER TO FB_HwRefInkStatDriveCover;
	bExecute		: BOOL;
END_VAR
VAR_OUTPUT
	bBusy		: BOOL;
	bError		: BOOL;
	nErrorId	: ERRORID;
END_VAR
VAR
	fbSdoWrite	: FB_SDO_WRITE;
	fbPower		: FB_CANOpenMotionPower;
	nState		: USINT;
	
	nStateA 		: USINT;
	nStateANext 	: USINT;
	bCancel			: BOOL;
	
	dwSdoIndex 		: DWORD;
	dwSdoSubIndex 	: DWORD;
	dwSdoDataLength : DWORD;
	nSdoDataValue 	: DINT;
	
END_VAR

IF bExecute THEN
	CASE nState OF
		0:	//Prepare
			bBusy := TRUE;
			pDriveRef^.P_eCoverState := E_OpClState.UNDEFINED;
			pDriveRef^.bIsInit := FALSE;
			A_Prepare();
			IF nStateA >= 80 THEN
				IF nStateA >= 99 THEN
					bError := TRUE;
					bBusy := FALSE;
					nState := 99;
				ELSE
					IF bCancel THEN
						nState := 80;
						bBusy := FALSE;
					ELSE
						nState := 1;	
					END_IF
				END_IF
				nStateA := 0;
			END_IF

		1:	//PowerOn
			fbPower(pControl:= ADR(pDriveRef^.nControl), pStatus:= ADR(pDriveRef^.nStatus), bExecute:= TRUE);
			IF NOT 	fbPower.bBusy THEN
				IF fbPower.bError THEN
					bError := TRUE;
					bBusy := FALSE;
					nState := 99;
				ELSE
					pDriveRef^.bDigiOut1 := TRUE;	//Versorgung für Digitale IOs (5V) einschalten
					pDriveRef^.nOpMode := 6; 		//Mode = Homing-Mode
					nState := 2;
				END_IF
				fbPower(bExecute:= FALSE);
			END_IF
			IF bCancel THEN
				fbPower(bExecute:= FALSE);
				bBusy := FALSE;	
			END_IF			
			
		2:	//Homing
			IF bCancel THEN
				nState := 70;
			END_IF
			pDriveRef^.nControl := 31;
			IF pDriveRef^.nStatus.3 OR pDriveRef^.nStatus.13 THEN //Error
				nState := 99;
			ELSIF NOT pDriveRef^.nStatus.10 AND NOT pDriveRef^.nStatus.12 AND NOT pDriveRef^.nStatus.13 THEN //Homing in process
				nState := 3;
			END_IF
			IF bCancel THEN
				nState := 70;
			END_IF
			
		3:	//Homing ready?
			IF pDriveRef^.nStatus.3 OR pDriveRef^.nStatus.13 THEN //Error
				nState := 99;
			ELSIF (pDriveRef^.nStatus AND 16#1400) = 16#1400 THEN
				pDriveRef^.nControl := 15;
			 	pDriveRef^.nOpMode := 1;
				pDriveRef^.bIsInit := TRUE;
				pDriveRef^.P_eCoverState := E_OpClState.Closed;
				bBusy := FALSE;
			END_IF
			IF bCancel THEN
				nState := 70;
			END_IF
			
		70:	//Homing stoppen
			pDriveRef^.nControl := 15;
			nState := 80;
			bBusy := FALSE;
	END_CASE
ELSE
	bError := FALSE;
	bCancel := FALSE;
	nErrorId := 0;
	nState := 0;
END_IF

ACTION A_Prepare:
CASE nStateA OF
	0:	//Errorbit gesetzt?
			IF pDriveRef^.nStatus.3 THEN //Error zurücksetzen
				pDriveRef^.nControl := 153;
			ELSE
				pDriveRef^.nControl := 0;
				nStateA := 1;
			END_IF
			
	1:	//SwitchParameters setzen (keine Endlagen verwenden)		
		dwSdoIndex := 16#2005;
		dwSdoSubIndex := 0;
		dwSdoDataLength := 4;
		nSdoDataValue := 3; //keine Endlagen
		nStateANext := 2;
		nStateA := 60; //Sdo senden			
			
	2:	//Brake deaktivieren
		dwSdoIndex := 16#200C;
		dwSdoSubIndex := 2;
		dwSdoDataLength := 1;
		nSdoDataValue := 0; //keine Brake
		nStateANext := 3;
		nStateA := 60; //Sdo senden

	3:	//Digital Outputmask setzen		
		dwSdoIndex := 16#2703;
		dwSdoSubIndex := 2;
		dwSdoDataLength := 4;
		nSdoDataValue := 16#30000; //Mask
		nStateANext := 4;
		nStateA := 60; //Sdo senden
		
	4:	//Fast Homing Speed setzen
		dwSdoIndex := 16#6099;
		dwSdoSubIndex := 1;
		dwSdoDataLength := 4;
		nSdoDataValue := 400; //Speed
		nStateANext := 5;
		nStateA := 60; //Sdo senden		

	5:	//Fast Homing Speed setzen
		dwSdoIndex := 16#6099;
		dwSdoSubIndex := 2;
		dwSdoDataLength := 4;
		nSdoDataValue := 100; //Speed
		nStateANext := 6;
		nStateA := 60; //Sdo senden		
		
	6:	//Profile Speed setzen		
		dwSdoIndex := 16#6081;
		dwSdoSubIndex := 0;
		dwSdoDataLength := 4;
		nSdoDataValue := 1200; //Speed
		nStateANext := 7;
		nStateA := 60; //Sdo senden		

	7:	//Homing Method setzen		
		dwSdoIndex := 16#6098;
		dwSdoSubIndex := 0;
		dwSdoDataLength := 1;
		nSdoDataValue := 19; //Method
		nStateANext := 8;
		nStateA := 60; //Sdo senden		

	8:	//Position Window setzen		
		dwSdoIndex := 16#6067;
		dwSdoSubIndex := 0;
		dwSdoDataLength := 4;
		nSdoDataValue := 100; //Window
		nStateANext := 80;
		nStateA := 60; //Sdo senden		
			
	60:	//Send SDO
		fbSdoWrite(sADSNetID:= pDriveRef^.stAdsAdress.sNetId,nPortNr:= pDriveRef^.stAdsAdress.nPort, 
					nIndex:= dwSdoIndex, nSubIndex:= dwSdoSubIndex, nDataLength:= dwSdoDataLength,
					 nData:= nSdoDataValue, bExecute:= TRUE);
		IF NOT fbSdoWrite.bBusy THEN
			IF fbSdoWrite.bError THEN
				nErrorId := fbSdoWrite.nAdsErrorId;
				nStateA := 99;
			ELSE
				nStateA := nStateANext;
			END_IF
			fbSdoWrite(bExecute:= FALSE);
		END_IF	
END_CASE
END_ACTION

METHOD M_Stop
VAR_INPUT
END_VAR
IF bBusy THEN
	bCancel := TRUE;	
END_IF
END_METHOD

END_FUNCTION_BLOCK

// ---- Hardware/InkStation/FB_InkStationOpenClose.TcPOU
FUNCTION_BLOCK FB_InkStationOpenClose
VAR_INPUT
	pDriveRef		: POINTER TO FB_HwRefInkStatDriveCover;
	eCtrl			: E_OpClCtrl;
	bExecute		: BOOL;	
END_VAR
VAR_OUTPUT
	bBusy		: BOOL;
	bError		: BOOL;
	nErrorId	: ERRORID;	
END_VAR
VAR
	nState		: USINT;
	timer		: TON;
END_VAR

IF bExecute THEN
	CASE nState OF
		0:
			IF pDriveRef = 0 THEN
				bError := TRUE;
				RETURN;		
			END_IF
			nState := 1;
			bBusy := TRUE;
			pDriveRef^.P_eCoverState := E_OpClState.UNDEFINED;
			IF NOT pDriveRef^.bIsInit THEN
				bBusy := FALSE;
				bError:= TRUE;
				nErrorId := E_ErrorIdCmd.ERRORID_DeviceNotInitialized;
				nState := 99;
			ELSE
				IF eCtrl = E_OpClCtrl.Open THEN
					pDriveRef^.nTargetPos := 102000;
				ELSE
					pDriveRef^.nTargetPos := -14000;
				END_IF
				pDriveRef^.nControl := 31;
			END_IF
			
		1:	//Warten auf Setpoint ACK
			timer(IN:=TRUE, PT:= T#100MS);
			IF pDriveRef^.nStatus.12 THEN
				timer(IN:=FALSE);
				pDriveRef^.nControl := 15;
				nState := 2;
			END_IF
			IF timer.Q THEN
				bBusy := FALSE;
				bError := TRUE;
				nErrorId := E_ErrorIdMultiZ.ERRORID_ToWaitSetPointAck;
				nState := 99;
			END_IF
			
		2:	//Warten auf Target reached
			timer(IN:=TRUE, PT:= T#5S);
			IF pDriveRef^.nStatus.10 THEN
				bBusy := FALSE;
				timer(IN:= FALSE);
				//Abfrage auf Endschalter
				IF eCtrl = E_OpClCtrl.Open THEN //Öffnen
					pDriveRef^.P_eCoverState := E_OpClState.Open;
					IF NOT pDriveRef^.bOpenSwitch THEN
						pDriveRef^.P_eCoverState := E_OpClState.UNDEFINED;
						bError := TRUE;
						nErrorId := E_ErrorIdCmd.ERRORID_CoverNotOpen;
						nState := 99; //Error, Deckel nicht richtig offen
					END_IF
				ELSE //Schließen
					pDriveRef^.P_eCoverState := E_OpClState.Closed;
					IF NOT pDriveRef^.bClosedSwitch THEN
						pDriveRef^.P_eCoverState := E_OpClState.UNDEFINED;
						bError := TRUE;
						nErrorId := E_ErrorIdCmd.ERRORID_CoverNotClosed;
						nState := 99; //Error, Deckel nicht richtig geschlossen
					END_IF
				END_IF
			END_IF
			IF timer.Q THEN
				bBusy := FALSE;
				bError := TRUE;
				nErrorId := E_ErrorIdMultiZ.ERRORID_ToWaitTrgtReached;
				nState := 99;
			END_IF
	END_CASE
ELSE
	bError := FALSE;
	nState := 0;
	nErrorId := 0;
	timer(IN:= FALSE);
END_IF

END_FUNCTION_BLOCK

// ---- Objects/Tools/FB_StampSupport.TcPOU
FUNCTION_BLOCK FB_StampSupport EXTENDS FB_MzTool
VAR_INPUT
END_VAR
VAR_OUTPUT
END_VAR
VAR
	
	//Specproperties
	rZOffsetUnlocked		: REAL;
	rZOffsetLocked			: REAL;
	
	pPneuChannelPress		: POINTER TO FB_PneuChannelRef;
	pPneuChannelVac			: POINTER TO FB_PneuChannelRef;
	
	nDOutChanValvePress		: USINT;	//Digitaler Ausgangskanal MzHead Druckventil
	nDOutChanValveVac		: USINT;	//Digitaler Ausgangskanal MzHead Vakuumventil
	fbMultiZStamp			: FB_MultiZStamp;
	
	//****************************************Aktionsvariablen****************************************************
	
	//Action: "InitTool"
	bInitTool			: BOOL;
	bInitSpecFlag		: BOOL := TRUE;
	nStateA_InitTool	: USINT;
	
	//Action: "SetPressure"
	bSetPress			: BOOL;
	fbSetPress			: FB_SetPressure;

	//Action: "SetVacuum"
	bSetVacuum			: BOOL;
	fbSetVacuum			: FB_SetPressure;
	
	//Action: "SwitchPressure"
	bSwitchPress		: BOOL;
	nStateA_SwitchPress	: USINT;		//State von A_SwitchPress()
	bPressOn			: BOOL;			//Druckventil "Auf"
	ePressCtrl			: E_PressCtrl;
	tPressTime			: TIME;			//Öffnungszeit Druckventil
	timerPress			: TON;			//Timer für Öffnungszeit Druckventil

	//Action: "PulsePressure"
	bPulsePress			: BOOL;
	nStateA_PulsePress	: USINT;	//State von A_PulsePress()
	eSwitchCtrlPhase1	: E_PressCtrl;		//
	eSwitchCtrlPhase2	: E_PressCtrl;		//
	nPulseDutycycle		: UINT;		//Tastverhältnis (0-100%)
	nTimePhase1			: UINT;
	nTimePhase2			: UINT;
	timerPulse			: TON;		//Timer
	nSetpointPulses		: UINT;		//Soll Anzahl an Pulses
	nCurrentPulses		: UINT;		//aktuelle Anzahl an Pulses
	bPulseOn			: BOOL;
	
	//Action: "LockUnlock"
	bLockUnlock				: BOOL;
	nStateA_LockUnlock		: USINT;	//State von A_LockUnlock
	bLock					: BOOL;		//True = Verriegeln, False = Entriegeln
	
	//Action: "Adjust"
	bAdjust					: BOOL;
	nStateA_Adjust			: USINT;	//State von A_Adjust
	nAdjustAngle			: INT;		//absolute Winkeleinstellung in 1/1000°	
	
	//Action: "Expose"
	bExpose					: BOOL;
	nStateA_Expose			: USINT;	//State von A_Expose
	bExposeStart			: BOOL;
	timerExpose				: TON;
	//bDigiOut				AT %Q* : BOOL;

	eCurPressState			: E_PressCtrl;
	nCurPressValue			: INT;
	
END_VAR

IF eCurrentState = E_MachineState.MACHINESTATE_Active THEN
	IF bInitTool THEN
		A_InitTool();
		IF nStateA_InitTool >= 80 THEN
			IF nStateA_InitTool >= 99 THEN
				bError := TRUE;
			END_IF
			bInitTool := FALSE;
			nStateA_InitTool := 0;
			M_RemoveListEntry(nSearchValue:= E_Action.ACTION_Init);
		END_IF		
	END_IF

	IF bLockUnlock THEN
		A_LockUnlock();
		IF nStateA_LockUnlock >= 80 THEN
			IF nStateA_LockUnlock >= 99 THEN
				bError := TRUE;		
			END_IF
			bLockUnlock := FALSE;
			nStateA_LockUnlock := 0;
			M_RemoveListEntry(nSearchValue:= E_Action.ACTION_LockUnlock);
		END_IF
	END_IF
	
	IF bSetPress THEN
		fbSetPress(pPneuChannelRef:= pPneuChannelPress);
		IF NOT fbSetPress.bBusy THEN
			IF fbSetPress.bError THEN
				bError := TRUE;
				stError.ErrorId := fbSetPress.nErrorId;
				stError.POU := E_POU.POU_FB_StampSupport;
				fbErrorList.M_Add(stError);
			END_IF
			bSetPress := FALSE;
			fbSetPress(pPneuChannelRef:= pPneuChannelPress, bExecute:= FALSE);
			M_RemoveListEntry(nSearchValue:= E_Action.ACTION_SetPressure);
		END_IF
	END_IF	

	IF bSetVacuum THEN
		fbSetVacuum(pPneuChannelRef:= pPneuChannelVac);
		IF NOT fbSetVacuum.bBusy THEN
			IF fbSetVacuum.bError THEN
				bError := TRUE;
				stError.ErrorId := fbSetVacuum.nErrorId;
				stError.POU := E_POU.POU_FB_StampSupport;
				fbErrorList.M_Add(stError);
			END_IF
			bSetVacuum := FALSE;
			fbSetVacuum(pPneuChannelRef:= pPneuChannelVac, bExecute:= FALSE);
			M_RemoveListEntry(nSearchValue:= E_Action.ACTION_SetVacuum);
		END_IF
	END_IF	
	
	IF bSwitchPress THEN
		A_SwitchPress();
		IF nStateA_SwitchPress >= 80 THEN
			IF nStateA_SwitchPress >= 99 THEN
				bError := TRUE;
			END_IF
			bSwitchPress := FALSE;
			nStateA_SwitchPress := 0;
			M_RemoveListEntry(nSearchValue:= E_Action.ACTION_SwitchPressure);
		END_IF
	END_IF	

	IF bPulsePress THEN	//Druck/Vakuum Ein/Aus
		A_PulsePress();
		IF nStateA_PulsePress >= 80 THEN
			IF nStateA_PulsePress >= 99 THEN
				bError := TRUE;
			END_IF
			bPulsePress := FALSE;
			nStateA_PulsePress := 0;
			M_RemoveListEntry(nSearchValue:= E_Action.ACTION_PulsePressure);
		END_IF
	END_IF
	
	IF bAdjust THEN
		A_Adjust();
		IF nStateA_Adjust >= 80 THEN
			IF nStateA_Adjust >= 99 THEN
				bError := TRUE;
			END_IF
			bAdjust := FALSE;
			nStateA_Adjust := 0;
			M_RemoveListEntry(nSearchValue:= E_Action.ACTION_StampAdjust);
		END_IF
	END_IF
	
	IF bExpose THEN
		A_Expose();
		IF nStateA_Expose >= 80 THEN
			IF nStateA_Expose >= 99 THEN
				bError := TRUE;
			END_IF
			bExpose := FALSE;
			nStateA_Expose := 0;
			M_RemoveListEntry(nSearchValue:= E_Action.ACTION_Expose);
		END_IF
	END_IF
	
END_IF

fbMultiZStamp(pFbMultiZ := pFbMultiZ);

SUPER^();	//FB_MzTool aufrufen

//Prozessdaten aktualisieren

stProcessData.n32Data[7].0 := pFbMultiZ^.stStampSupport.bLocked;
stProcessData.n32Data[7].1 := pFbMultiZ^.stStampSupport.bLight;
stProcessData.n32Data[7].2 := pFbMultiZ^.stStampSupport.bStampInSupport;
stProcessData.n32Data[7].3 := GVL_HwRefIO.bTrigger1;

IF pFbMultiZ^.stStampSupport.bAngleReached THEN
	stProcessData.n32Data[8] := pFbMultiZ^.stStampSupport.nAngleSetpoint;
END_IF

IF pPneuChannelPress > 0 THEN
	stProcessData.n32Data[9] := pPneuChannelPress^.P_nSetPressure;
	stProcessData.n32Data[10] := pPneuChannelPress^.P_nCurrentPressure;
	nCurPressValue := pPneuChannelPress^.P_nCurrentPressure;
END_IF

IF pPneuChannelVac > 0 THEN
	stProcessData.n32Data[11] := pPneuChannelVac^.P_nSetPressure;
	stProcessData.n32Data[12] := pPneuChannelVac^.P_nCurrentPressure;
END_IF

IF pFbMultiZ > 0 THEN
	IF NOT (pFbMultiZ^.aDigiOut[nDOutChanValvePress] OR pFbMultiZ^.aDigiOut[nDOutChanValveVac]) THEN
		eCurPressState := E_PressCtrl.PRESSCTRL_Off;
	ELSIF pFbMultiZ^.aDigiOut[nDOutChanValvePress] AND NOT pFbMultiZ^.aDigiOut[nDOutChanValveVac] THEN
		eCurPressState := E_PressCtrl.PRESSCTRL_PressOn;
	ELSIF NOT pFbMultiZ^.aDigiOut[nDOutChanValvePress] AND pFbMultiZ^.aDigiOut[nDOutChanValveVac] THEN
		eCurPressState := E_PressCtrl.PRESSCTRL_VacOn;	
	ELSE
		eCurPressState := E_PressCtrl.PRESSCTRL_UNDEFINED;
	END_IF
END_IF

stProcessData.n32Data[13] := eCurPressState;
aObjProcData[nNotifyId] := stProcessData;

PROPERTY P_rZOffsetLocked : REAL
GET
P_rZOffsetLocked := rZOffsetLocked;
END_GET
END_PROPERTY

METHOD M_GetAllProps : ERRORID
VAR_INPUT
	refCmdData : REFERENCE TO  ST_CmdData;
END_VAR
//Basisproperties lesen
SUPER^.M_GetAllProps(refCmdData);
//Specialproperties lesen
nCurrentPropIndex := nCurrentPropIndex + 1;
refCmdData.n32Data[nCurrentPropIndex] := REAL_TO_DINT(rZOffsetUnlocked);
nCurrentPropIndex := nCurrentPropIndex + 1;
refCmdData.n32Data[nCurrentPropIndex] := REAL_TO_DINT(rZOffsetLocked);

nCurrentPropIndex := nCurrentPropIndex + 1;
IF pPneuChannelPress > 0 THEN
	refCmdData.n32Data[nCurrentPropIndex] := pPneuChannelPress^.nChannel;
ELSE
	refCmdData.n32Data[nCurrentPropIndex] := 0;
END_IF

nCurrentPropIndex := nCurrentPropIndex + 1;
IF pPneuChannelVac > 0 THEN
	refCmdData.n32Data[nCurrentPropIndex] := pPneuChannelVac^.nChannel;
ELSE
	refCmdData.n32Data[nCurrentPropIndex] := 0;
END_IF

nCurrentPropIndex := nCurrentPropIndex + 1;
refCmdData.n32Data[nCurrentPropIndex] := nDOutChanValvePress; //Digitaler Ausgangskanal MzHead Druckventil
nCurrentPropIndex := nCurrentPropIndex + 1;
refCmdData.n32Data[nCurrentPropIndex] := nDOutChanValveVac; //Digitaler Ausgangskanal MzHead Vakuumventil
END_METHOD

PROPERTY P_bStampInMagazine : BOOL
GET
P_bStampInMagazine := fbMultiZStamp.P_bStampInMagazine;
END_GET
END_PROPERTY

METHOD M_GetPressValueOk : BOOL
VAR_INPUT
	nSetPressure	: INT;
	nTolerancePlus	: INT;
	nToleranceMinus	: INT;
END_VAR
IF (nCurPressValue >= nSetPressure - nToleranceMinus) AND (nCurPressValue <= nSetPressure + nTolerancePlus)THEN
	M_GetPressValueOk := TRUE;
	RETURN;
END_IF
END_METHOD

PROPERTY P_bIsInit : BOOL
GET
P_bIsInit := bInitToolOk AND SUPER^.P_bIsInit;
END_GET
END_PROPERTY

ACTION A_SwitchPress:
CASE nStateA_SwitchPress OF
	0:
		timerPress(IN:= TRUE, PT:= tPressTime);
		nStateA_SwitchPress := 1;
		
	1:	//Warten bis Zeitabgelaufen
		timerPress();
		IF timerPress.Q THEN
			timerPress(IN:= FALSE);
			pFbMultiZ^.aDigiOut[nDOutChanValvePress] := FALSE;
			pFbMultiZ^.aDigiOut[nDOutChanValveVac] := FALSE;
			nStateA_SwitchPress := 80;
		END_IF
		
	70:	//Abbrechen
		timerPress(IN:= FALSE);
		nStateA_SwitchPress := 80;
END_CASE
END_ACTION

PROPERTY P_bLocked : BOOL
GET
P_bLocked := pFbMultiZ^.stStampSupport.bLocked;
END_GET
END_PROPERTY

PROPERTY P_nCurPressValue : INT
GET
P_nCurPressValue := nCurPressValue;
END_GET
END_PROPERTY

ACTION A_Expose:
CASE nStateA_Expose OF
	0:	
		GVL_HwRefIO.bTrigger1 := TRUE;
		//Timer starten
		IF timerExpose.PT > T#0S THEN
			timerExpose(IN:=TRUE);
			nStateA_Expose := 1;
		ELSE
			nStateA_Expose := 2;
		END_IF
	
	1:	//Warten, bis Zeit abgelaufen
		timerExpose();
		IF timerExpose.Q THEN
			timerExpose(IN:= FALSE);
			GVL_HwRefIO.bTrigger1 := FALSE;
			nStateA_Expose := 2;
		END_IF
		
	2:	//Delay bis ready (Blendenschaltzeit)
		timerExpose(IN:=TRUE,PT:=T#500MS);
		IF timerExpose.Q THEN
			timerExpose(IN:=FALSE);
			nStateA_Expose := 80;
		END_IF	
		
	70:	//Abbrechen
		timerExpose(IN:= FALSE);
		GVL_HwRefIO.bTrigger1 := FALSE;
		nStateA_Expose := 80;
END_CASE
END_ACTION

METHOD M_CheckAction : ERRORID
VAR_INPUT
	refActionData 	: REFERENCE TO ST_ActionData;
	pCorrelObject	: POINTER TO FB_Object;
END_VAR

VAR
	pStampMagazine : POINTER TO FB_StampMagazine;
END_VAR
CASE refActionData.eAction OF
	E_Action.ACTION_MoveToTarget:
		M_CheckAction := SUPER^.M_CheckAction(refActionData,pCorrelObject);
		IF M_CheckAction > 0 THEN
			RETURN;
		END_IF
		IF fbMultiZStamp.P_bStampInSupport THEN	//Sensor zeigt an, dass Stamp aufgenommen
			IF pPiece = 0 THEN
				M_CheckAction := E_ErrorIdCmd.ERRORID_InvalidStampAssignment;
			END_IF
		ELSE
			IF pPiece > 0 THEN
				M_CheckAction := E_ErrorIdCmd.ERRORID_InvalidStampAssignment;
			END_IF
		END_IF

	E_Action.ACTION_ExchangePiece:
		IF fbObjectDirectory.M_GetObjType(refActionData.nTarget) <> E_ObjectType.OBJECTTYPE_StampMagazine THEN
			M_CheckAction := E_ErrorIdCmd.ERRORID_UnsuitableTarget;
		ELSE
			IF refActionData.aParams[2] = 0 THEN //Drop - es muss ein Stamp im Support sein
				IF pPiece = 0 OR NOT P_bStampInSupport THEN
					M_CheckAction := E_ErrorIdCmd.ERRORID_NoPieceOnTool;
				END_IF
			ELSIF refActionData.aParams[2] = 1 THEN //Take - es darf kein Stamp im Support sein
				IF pPiece > 0 OR P_bStampInSupport THEN 
					M_CheckAction := E_ErrorIdCmd.ERRORID_PieceAlreadyOnTool;	
				END_IF
			ELSE
				M_CheckAction := E_ErrorIdCmd.ERRORID_InvalidCtrl;
			END_IF
		END_IF
	E_Action.ACTION_MeasureTool:
		IF fbObjectDirectory.M_GetObjType(refActionData.nTarget) = E_ObjectType.OBJECTTYPE_InkStation THEN
			;
		ELSIF fbObjectDirectory.M_GetObjType(refActionData.nTarget) = E_ObjectType.OBJECTTYPE_StampMagazine THEN
			pStampMagazine := fbObjectDirectory.M_GetObjPointer(refActionData.nTarget);
			//Ist der MeasurePoint vorhanden?
			IF NOT pStampMagazine^.P_bMeasurePointAvailable THEN
				M_CheckAction := E_ErrorIdCmd.ERRORID_UnsuitableTarget;	
			END_IF
		ELSE
			M_CheckAction := E_ErrorIdCmd.ERRORID_UnsuitableTarget;
		END_IF
		//Es muss ein Stempel im Support sein
		IF NOT (P_bStampInSupport AND pPiece > 0) THEN
			M_CheckAction := E_ErrorIdCmd.ERRORID_NoPieceOnTool;
		END_IF
		
	E_Action.ACTION_Expose, //BasicAction für ActionOnArray
	E_Action.ACTION_SwitchPressure: //BasicAction für ActionOnArray
	E_Action.ACTION_StampInking,
	E_Action.ACTION_StampDemolding:
		IF pPiece = 0 THEN
			M_CheckAction := E_ErrorIdCmd.ERRORID_NoPieceOnTool;
		END_IF		
ELSE
	M_CheckAction := SUPER^.M_CheckAction(refActionData, pCorrelObject);
END_CASE
END_METHOD

ACTION A_Stop:
IF nStateA_Stop = 0 THEN

	IF bInitTool AND nStateA_InitTool < 70 THEN
		nStateA_InitTool := 70;
	END_IF
	
	IF bSetPress THEN
		fbSetPress(bExecute:= FALSE, pPneuChannelRef:= pPneuChannelPress);
	END_IF

	IF bSetVacuum THEN
		fbSetVacuum(bExecute:= FALSE, pPneuChannelRef:= pPneuChannelVac);
	END_IF
	
	IF bSwitchPress AND nStateA_SwitchPress < 70 THEN
		nStateA_SwitchPress := 70;
	END_IF

	IF bLockUnlock AND nStateA_LockUnlock < 70 THEN
		nStateA_LockUnlock := 70;
	END_IF
	
	IF bExpose AND nStateA_Expose < 70 THEN
		nStateA_Expose := 70;
	END_IF
	
	IF bPulsePress AND nStateA_PulsePress < 70 THEN
		nStateA_PulsePress := 70;
	END_IF

	nStateA_Stop := 1;
END_IF

SUPER^.A_Stop();
END_ACTION

ACTION A_InitTool:
IF nStateA_InitTool > 0 AND fbMultiZStamp.bError THEN
	stError.ErrorId := fbMultiZStamp.nErrorId;
	stError.POUState := nStateA_InitTool;
	nStateA_InitTool := 99;
END_IF

CASE nStateA_InitTool OF
	0:	//Warten bis InitBase fertig
		IF NOT bInitAxis THEN
			bInitToolOk := FALSE;
			IF bError THEN
				nStateA_InitTool := 0;
				bInitTool := FALSE;
				M_RemoveListEntry(nSearchValue:= E_Action.ACTION_Init);
				RETURN;
			END_IF
			nStateA_InitTool := 1;
		END_IF
		
	1:	//Stamp initialisieren
		fbMultiZStamp.M_Init();
		nStateA_InitTool := 2;
		
	2:	//Warten bis Initialisierung fertig
		IF NOT fbMultiZStamp.bBusy THEN
			bInitToolOk := TRUE;
			nStateA_InitTool := 80;
		END_IF
		
	70:	//Abbrechen
		fbMultiZStamp.M_Stop();
		nStateA_InitTool := 71;
		
	71:	
		IF NOT fbMultiZStamp.bBusy THEN
			nStateA_InitTool := 80;
		END_IF
		
END_CASE

//Errorhandling
IF nStateA_InitTool = 99 THEN
	stError.POU := E_POU.POU_FB_StampSupport;
	stError.Cmd := E_Action.ACTION_Init;
	stError.POUAction := E_POUACT.POUACT_A_InitSpec;
	fbErrorList.M_Add(stError);
END_IF
END_ACTION

METHOD M_ExeAction : ERRORID
VAR_INPUT
	refActionData : REFERENCE TO ST_ActionData;	
END_VAR
IF NOT (eCurrentState = E_MachineState.MACHINESTATE_Idle OR
	eCurrentState = E_MachineState.MACHINESTATE_Active OR
	eCurrentState = E_MachineState.MACHINESTATE_Ready) THEN
	M_ExeAction := E_ErrorIdCmd.ERRORID_InvalidState;
	RETURN;
END_IF

CASE refActionData.eAction OF
	E_Action.ACTION_Init:
		IF NOT bInitAxis AND NOT bInitTool THEN
			bInitAxis := TRUE;
			bInitTool := TRUE;
			fbList.A_AddHeadValue( hList := hList, putValue := E_Action.ACTION_Init);	//InitAxis
			fbList.A_AddHeadValue( hList := hList, putValue := E_Action.ACTION_Init);	//InitTool
		ELSE
			RETURN;
		END_IF	

	E_Action.ACTION_LockUnlock:
		IF NOT bLockUnlock THEN
			bLockUnlock := TRUE;
			bLock := DINT_TO_BOOL(refActionData.aParams[1]);		
			fbList.A_AddHeadValue( hList := hList, putValue := E_Action.ACTION_LockUnlock); 
		END_IF
		
	E_Action.ACTION_SetPressure:
		fbSetPress(bExecute:= FALSE, pPneuChannelRef:= pPneuChannelPress); //eventueller Fehler wird auch zurückgesetzt
		fbSetPress.bAwait := DINT_TO_BOOL(refActionData.aParams[1]);
		fbSetPress.nValue := DINT_TO_INT(refActionData.aParams[2]);
		fbSetPress.nTolerancePlus := DINT_TO_INT(refActionData.aParams[3]);
		fbSetPress.nToleranceMinus := DINT_TO_INT(refActionData.aParams[4]);
		fbSetPress.tTimeout := DINT_TO_TIME(refActionData.aParams[5]);
		
		fbSetPress(bExecute:= TRUE,	pPneuChannelRef:= pPneuChannelPress,nErrorId=> M_ExeAction);
		IF fbSetPress.bError THEN
			RETURN;
		END_IF
		
		IF NOT bSetPress AND fbSetPress.bBusy THEN
			bSetPress := TRUE;
			fbList.A_AddHeadValue(hList := hList, putValue := E_Action.ACTION_SetPressure);
		ELSE
			RETURN;	
		END_IF

	E_Action.ACTION_SetVacuum:
		fbSetVacuum(bExecute:= FALSE, pPneuChannelRef:= pPneuChannelVac); //eventueller Fehler wird auch zurückgesetzt
		fbSetVacuum.bAwait := DINT_TO_BOOL(refActionData.aParams[1]);
		fbSetVacuum.nValue := DINT_TO_INT(refActionData.aParams[2]);
		fbSetVacuum.nTolerancePlus := DINT_TO_INT(refActionData.aParams[3]);
		fbSetVacuum.nToleranceMinus := DINT_TO_INT(refActionData.aParams[4]);
		fbSetVacuum.tTimeout := DINT_TO_TIME(refActionData.aParams[5]);
		
		fbSetVacuum(bExecute:= TRUE, pPneuChannelRef:= pPneuChannelVac,nErrorId=> M_ExeAction);
		IF fbSetVacuum.bError THEN
			RETURN;
		END_IF
		
		IF NOT bSetVacuum AND fbSetVacuum.bBusy THEN
			bSetVacuum := TRUE;
			fbList.A_AddHeadValue(hList := hList, putValue := E_Action.ACTION_SetVacuum);
		ELSE
			RETURN;	
		END_IF
		
	E_Action.ACTION_SwitchPressure:
		//Pneumatikkanal checken
		ePressCtrl := DINT_TO_USINT(refActionData.aParams[1]);
		tPressTime := DINT_TO_TIME(refActionData.aParams[2]);
		CASE ePressCtrl OF
			E_PressCtrl.PRESSCTRL_Off:
				pFbMultiZ^.aDigiOut[nDOutChanValvePress] := FALSE;
				pFbMultiZ^.aDigiOut[nDOutChanValveVac] := FALSE;
				RETURN;			
			E_PressCtrl.PRESSCTRL_PressOn:
				pFbMultiZ^.aDigiOut[nDOutChanValvePress] := TRUE;
				pFbMultiZ^.aDigiOut[nDOutChanValveVac] := FALSE;
				IF tPressTime = T#0S THEN
					RETURN;			
				ELSE
					bSwitchPress := TRUE;
					fbList.A_AddHeadValue(hList := hList, putValue := E_Action.ACTION_SwitchPressure);					
				END_IF
			E_PressCtrl.PRESSCTRL_VacOn:
				pFbMultiZ^.aDigiOut[nDOutChanValvePress] := FALSE;
				pFbMultiZ^.aDigiOut[nDOutChanValveVac] := TRUE;
				IF tPressTime = T#0S THEN
					RETURN;					
				ELSE
					bSwitchPress := TRUE;
					fbList.A_AddHeadValue(hList := hList, putValue := E_Action.ACTION_SwitchPressure);					
				END_IF
		ELSE
			RETURN;
		END_CASE
		
	E_Action.ACTION_PulsePressure:
		bPulseOn := DINT_TO_BOOL(refActionData.aParams[6]);
		IF bPulseOn THEN	//On
			eSwitchCtrlPhase1 := DINT_TO_USINT(refActionData.aParams[1]);
			eSwitchCtrlPhase2 := DINT_TO_USINT(refActionData.aParams[2]);
	
			IF NOT(refActionData.aParams[4] >= 1 AND refActionData.aParams[4] <= 100) THEN
				M_ExeAction := E_ErrorIdCmd.ERRORID_InvalidDutyCycle;  //Error
				RETURN;
			END_IF
			
			nTimePhase1 := DINT_TO_UINT(refActionData.aParams[3] / 100 * refActionData.aParams[4]); 
			nTimePhase2 := DINT_TO_UINT(refActionData.aParams[3] - nTimePhase1);
			
			IF NOT bPulsePress THEN
				bPulsePress := TRUE;
				fbList.A_AddHeadValue(hList := hList, putValue := E_Action.ACTION_PulsePressure);
			ELSE
				RETURN;
			END_IF
			
			nCurrentPulses := 0;
			nSetpointPulses := DINT_TO_UINT(refActionData.aParams[5]);
		ELSE
			RETURN;
		END_IF
		
	E_Action.ACTION_StampAdjust:
		IF NOT bAdjust THEN
			//überprüfen ob Sollwinkel in gültigen Grenzen !!NOCH IMPLEMENTIEREN!!
			nAdjustAngle := DINT_TO_INT(refActionData.aParams[1]);
			bAdjust := TRUE;
			fbList.A_AddHeadValue(hList := hList, putValue := E_Action.ACTION_StampAdjust);
		ELSE
			RETURN;
		END_IF
		
	E_Action.ACTION_Expose:
		bExposeStart := DINT_TO_BOOL(refActionData.aParams[1]);
		IF NOT bExpose AND bExposeStart THEN
			timerExpose.PT := DINT_TO_TIME(refActionData.aParams[3]);
			fbList.A_AddHeadValue( hList := hList, putValue := E_Action.ACTION_Expose);
			bExpose := TRUE;
		ELSIF bExpose AND NOT bExposeStart THEN
			nStateA_Expose := 70;
		ELSE
			GVL_HwRefIO.bTrigger1 := FALSE;
		END_IF

	E_Action.ACTION_SwitchLight:
		fbMultiZStamp.P_bLight := DINT_TO_BOOL(refActionData.aParams[1]);
		RETURN;

	ELSE
		M_ExeAction := SUPER^.M_ExeAction(refActionData);
		RETURN;
END_CASE

bBusy := TRUE;
eCurrentState := E_MachineState.MACHINESTATE_Active;
END_METHOD

METHOD M_ClearAllProps
VAR_INPUT
	bIgnoreParent : BOOL; //Es wird das gesamte OD gelöscht. -> Zeiger auf Parent nicht mehr gültig!
END_VAR
pPneuChannelPress := 0;
pPneuChannelVac := 0;
SUPER^.M_ClearAllProps(bIgnoreParent);
END_METHOD

ACTION A_Reset:
//Ist noch eine Aktion aktiv?
IF nStateA_ResetSpec = 0 THEN 
	
	IF bAdjust THEN
		bAdjust := FALSE;
		nStateA_Adjust := 0;
	END_IF

	IF bExpose THEN
		bExpose := FALSE;
		nStateA_Expose := 0;
	END_IF

	IF bLockUnlock THEN
		bLockUnlock := FALSE;
		nStateA_LockUnlock := 0;
	END_IF
	
	IF bSetPress THEN
		bSetPress := FALSE;
		fbSetPress(bExecute:= FALSE, pPneuChannelRef:= pPneuChannelPress);
	END_IF

	IF bSetVacuum THEN
		bSetVacuum := FALSE;
		fbSetVacuum(bExecute:= FALSE, pPneuChannelRef:= pPneuChannelVac);
	END_IF
	
	IF bSwitchPress THEN 
		bSwitchPress := FALSE;
		nStateA_SwitchPress := 0;
	END_IF
	
	IF bPulsePress THEN 
		bPulsePress := FALSE;
		nStateA_PulsePress := 0;
	END_IF
	
	fbMultiZStamp.M_Reset();
	
	nStateA_ResetSpec := 80;		
END_IF

SUPER^.A_Reset();
END_ACTION

METHOD M_AddChild : ERRORID
VAR_INPUT
	pObject : POINTER TO FB_Object;
	nSlotNr	: UINT;
	nIndex 	: INT;
END_VAR
//Kann folgende Objekt-Typen aufnehmen
//Stamp
IF pObject > 0 THEN
	IF pObject^.P_eObjectType = E_ObjectType.OBJECTTYPE_Stamp OR
		 	pObject^.P_eObjectType = E_ObjectType.OBJECTTYPE_Exposure OR 
			pObject^.P_eObjectType = E_ObjectType.OBJECTTYPE_DummyTool OR
			pObject^.P_eObjectType = E_ObjectType.OBJECTTYPE_Camera THEN
		M_AddChild := SUPER^.M_AddChild(pObject,nSlotNr,nIndex);
	ELSE
		M_AddChild := E_ErrorIdObjMgmt.ERRORID_InvalidParentObject;
	END_IF
ELSE
	M_AddChild := E_ErrorIdObjMgmt.ERRORID_InvalidParentObject;
END_IF
END_METHOD

METHOD M_SetAllProps : ERRORID
VAR_INPUT
	refCmdData : REFERENCE TO  ST_CmdData;
END_VAR

VAR
	nPneuChannel : USINT;
END_VAR
M_SetAllProps := SUPER^.M_SetAllProps(refCmdData);

IF M_SetAllProps = 0 THEN
	fbMultiZStamp(pFbMultiZ := pFbMultiZ);
ELSE
	RETURN;
END_IF

nCurrentPropIndex := nCurrentPropIndex + 1;
nSpecPropIndex := nCurrentPropIndex;
rZOffsetUnlocked := DINT_TO_REAL(refCmdData.n32Data[nCurrentPropIndex]);
nCurrentPropIndex := nCurrentPropIndex + 1;
rZOffsetLocked := DINT_TO_REAL(refCmdData.n32Data[nCurrentPropIndex]);

//PneuChannel Druck
nCurrentPropIndex := nCurrentPropIndex + 1;
nPneuChannel := DINT_TO_USINT(refCmdData.n32Data[nCurrentPropIndex]);
IF NOT (nPneuChannel > 0 AND nPneuChannel <= cNoOfPneuChannels) THEN
	M_SetAllProps := E_ErrorIdObjMgmt.ERRORID_InvalidPneuChannel;
	RETURN;	
END_IF
pPneuChannelPress := ADR(aFbPneuChannel[nPneuChannel]);

//PneuChannel Vakuum
nCurrentPropIndex := nCurrentPropIndex + 1;
nPneuChannel := DINT_TO_USINT(refCmdData.n32Data[nCurrentPropIndex]);		
IF NOT (nPneuChannel > 0 AND nPneuChannel <= cNoOfPneuChannels) THEN
	M_SetAllProps := E_ErrorIdObjMgmt.ERRORID_InvalidPneuChannel;
	RETURN;	
END_IF
pPneuChannelVac := ADR(aFbPneuChannel[nPneuChannel]);

nCurrentPropIndex := nCurrentPropIndex + 1;
nDOutChanValvePress := DINT_TO_USINT(refCmdData.n32Data[nCurrentPropIndex]);	//Digitaler Ausgangskanal MzHead Druckventil Pressure
IF NOT(nDOutChanValvePress > 0 AND nDOutChanValvePress <= 7) THEN
	M_SetAllProps := E_ErrorIdObjMgmt.ERRORID_InvalidMzDOutChannel;
	RETURN;
END_IF

nCurrentPropIndex := nCurrentPropIndex + 1;
nDOutChanValveVac := DINT_TO_USINT(refCmdData.n32Data[nCurrentPropIndex]);	//Digitaler Ausgangskanal MzHead Druckventil Vacuum
IF NOT(nDOutChanValveVac > 0 AND nDOutChanValveVac <= 7) THEN
	M_SetAllProps := E_ErrorIdObjMgmt.ERRORID_InvalidMzDOutChannel;
	RETURN;
END_IF

pZAxisRef^.eFixedToolType := E_MzToolType.TOOL_TYPE_Stamp;

nNoOfProps := nCurrentPropIndex + 1;
END_METHOD

METHOD M_SetSingleProp : ERRORID
VAR_INPUT
	refCmdData : REFERENCE TO  ST_CmdData;
END_VAR

VAR
	nPneuChannel : USINT;
END_VAR
IF nSpecPropIndex = refCmdData.aHeader[1] THEN //ZOffsetUnlocked
	rZOffsetUnlocked := DINT_TO_REAL(refCmdData.n32Data[0]);
	
ELSIF (nSpecPropIndex + 1) = refCmdData.aHeader[1] THEN //ZOffsetLocked
	rZOffsetLocked := DINT_TO_REAL(refCmdData.n32Data[0]);
	
ELSIF (nSpecPropIndex + 1) = refCmdData.aHeader[1] THEN //PneuChannel Druck
	nPneuChannel :=  DINT_TO_USINT(refCmdData.n32Data[0]);
	IF NOT (nPneuChannel > 0 AND nPneuChannel <= cNoOfPneuChannels) THEN
		M_SetSingleProp := E_ErrorIdObjMgmt.ERRORID_InvalidPneuChannel;
		RETURN;	
	END_IF
	pPneuChannelPress := ADR(aFbPneuChannel[nPneuChannel]);	
		
ELSIF (nSpecPropIndex + 1) = refCmdData.aHeader[1] THEN //PneuChannel Vakuum
	nPneuChannel :=  DINT_TO_USINT(refCmdData.n32Data[0]);
	IF NOT (nPneuChannel > 0 AND nPneuChannel <= cNoOfPneuChannels) THEN
		M_SetSingleProp := E_ErrorIdObjMgmt.ERRORID_InvalidPneuChannel;
		RETURN;	
	END_IF
	pPneuChannelVac := ADR(aFbPneuChannel[nPneuChannel]);

ELSIF (nSpecPropIndex + 1) = refCmdData.aHeader[1] THEN //Digitaler Ausgangskanal Kopfbasisplatine für Druckventil
	IF refCmdData.n32Data[0] < 1 OR refCmdData.n32Data[0] > 9 THEN
		M_SetSingleProp := E_ErrorIdObjMgmt.ERRORID_InvalidMzDOutChannel;
		RETURN;
	END_IF
	nDOutChanValvePress := DINT_TO_USINT(refCmdData.n32Data[0]);
	
ELSIF (nSpecPropIndex + 1) = refCmdData.aHeader[1] THEN //Digitaler Ausgangskanal Kopfbasisplatine für Vakuumventil
	IF refCmdData.n32Data[0] < 1 OR refCmdData.n32Data[0] > 9 THEN
		M_SetSingleProp := E_ErrorIdObjMgmt.ERRORID_InvalidMzDOutChannel;
		RETURN;
	END_IF
	nDOutChanValveVac := DINT_TO_USINT(refCmdData.n32Data[0]);
	
ELSE
	M_SetSingleProp := SUPER^.M_SetSingleProp(refCmdData);
END_IF
END_METHOD

PROPERTY P_eCurPressState : E_PressCtrl
GET
P_eCurPressState := eCurPressState;
END_GET
END_PROPERTY

ACTION A_PulsePress:
CASE nStateA_PulsePress OF
	0:	//Phase1
		IF eSwitchCtrlPhase1 = E_PressCtrl.PRESSCTRL_Off THEN
			pFbMultiZ^.aDigiOut[nDOutChanValvePress] := FALSE;
			pFbMultiZ^.aDigiOut[nDOutChanValveVac] := FALSE;
		ELSIF eSwitchCtrlPhase1 = E_PressCtrl.PRESSCTRL_PressOn THEN
			pFbMultiZ^.aDigiOut[nDOutChanValvePress] := TRUE;
			pFbMultiZ^.aDigiOut[nDOutChanValveVac] := FALSE;
		ELSIF eSwitchCtrlPhase1 = E_PressCtrl.PRESSCTRL_VacOn THEN
			pFbMultiZ^.aDigiOut[nDOutChanValvePress] := FALSE;
			pFbMultiZ^.aDigiOut[nDOutChanValveVac] := TRUE;
		END_IF

		timerPulse(IN:= TRUE, PT:= UINT_TO_TIME(nTimePhase1));
		IF timerPulse.Q THEN
			timerPulse(IN:= FALSE);
			nStateA_PulsePress := 1;
			nCurrentPulses := nCurrentPulses + 1;
		END_IF

	1:	//Phase2
		IF eSwitchCtrlPhase2 = E_PressCtrl.PRESSCTRL_Off THEN
			pFbMultiZ^.aDigiOut[nDOutChanValvePress] := FALSE;
			pFbMultiZ^.aDigiOut[nDOutChanValveVac] := FALSE;
		ELSIF eSwitchCtrlPhase2 = E_PressCtrl.PRESSCTRL_PressOn THEN
			pFbMultiZ^.aDigiOut[nDOutChanValvePress] := TRUE;
			pFbMultiZ^.aDigiOut[nDOutChanValveVac] := FALSE;
		ELSIF eSwitchCtrlPhase2 = E_PressCtrl.PRESSCTRL_VacOn THEN
			pFbMultiZ^.aDigiOut[nDOutChanValvePress] := FALSE;
			pFbMultiZ^.aDigiOut[nDOutChanValveVac] := TRUE;
		END_IF	

		timerPulse(IN:= TRUE, PT:= UINT_TO_TIME(nTimePhase2));
		IF timerPulse.Q THEN
			timerPulse(IN:= FALSE);
			IF nCurrentPulses = nSetpointPulses THEN
				pFbMultiZ^.aDigiOut[nDOutChanValvePress] := FALSE;
				pFbMultiZ^.aDigiOut[nDOutChanValveVac] := FALSE;
				nStateA_PulsePress := 80;
			ELSIF nSetpointPulses = 0 AND NOT bPulseOn THEN
				pFbMultiZ^.aDigiOut[nDOutChanValvePress] := FALSE;
				pFbMultiZ^.aDigiOut[nDOutChanValveVac] := FALSE;
				nStateA_PulsePress := 80;
			ELSE
				nStateA_PulsePress := 0;	
			END_IF
		END_IF
		
	70:	//Abbrechen	
		pFbMultiZ^.aDigiOut[nDOutChanValvePress] := FALSE;
		pFbMultiZ^.aDigiOut[nDOutChanValveVac] := FALSE;
		timerPulse(IN:= FALSE);
		nStateA_PulsePress := 80;
END_CASE
END_ACTION

PROPERTY P_rZOffsetUnlocked : REAL
GET
P_rZOffsetUnlocked := rZOffsetUnlocked;
END_GET
END_PROPERTY

METHOD FB_init : BOOL
VAR_INPUT
	bInitRetains : BOOL; // if TRUE, the retain variables are initialized (warm start / cold start)
	bInCopyCode : BOOL;  // if TRUE, the instance afterwards gets moved into the copy code (online change)
END_VAR
eObjectType := E_ObjectType.OBJECTTYPE_StampSupport;
eObjectGroup := E_ObjectGroup.OBJECTGROUP_MzTool OR E_ObjectGroup.OBJECTGROUP_Device;
END_METHOD

PROPERTY P_bStampInSupport : BOOL
GET
P_bStampInSupport := fbMultiZStamp.P_bStampInSupport;
END_GET
END_PROPERTY

ACTION A_Adjust:
IF nStateA_Adjust = 0 THEN
	fbMultiZStamp.M_Adjust(nAdjustAngle);
	nStateA_Adjust := 1;
END_IF

IF nStateA_Adjust = 1 THEN
	IF NOT fbMultiZStamp.bBusy THEN
		nStateA_Adjust := 80;	
	END_IF
	
	IF fbMultiZStamp.bError THEN
		stError.Cmd := E_Action.ACTION_StampAdjust;
		stError.ErrorId := fbMultiZStamp.nErrorId;
		stError.POU := E_POU.POU_FB_StampSupport;
		stError.POUAction := E_POUACT.POUACT_A_Adjust;
		stError.POUState := nStateA_Adjust;
		fbErrorList.M_Add(stError);
		fbMultiZStamp.M_Reset();
		nStateA_Adjust := 99;	
	END_IF	
END_IF
END_ACTION

ACTION A_LockUnlock:
IF nStateA_LockUnlock = 0 THEN
	fbMultiZStamp.M_LockUnLock(bLock);
		nStateA_LockUnlock := 1;
END_IF

IF nStateA_LockUnlock = 1 THEN
	IF NOT fbMultiZStamp.bBusy THEN
		nStateA_LockUnlock := 80;	
	END_IF
	
	IF fbMultiZStamp.bError THEN
		stError.ErrorId := fbMultiZStamp.nErrorId;
		stError.Cmd := E_Action.ACTION_LockUnlock;
		stError.POU := E_POU.POU_FB_StampSupport;
		stError.POUAction := E_POUACT.POUACT_A_LockUnlock;
		stError.POUState := nStateA_LockUnlock;
		fbErrorList.M_Add(stError);			
		fbMultiZStamp.M_Reset();
		nStateA_LockUnlock := 99;	
	END_IF	
END_IF

IF nStateA_LockUnlock = 70 THEN
	IF fbMultiZStamp.bBusy THEN
		fbMultiZStamp.M_Stop();
	END_IF
	nStateA_LockUnlock := 80;
END_IF
END_ACTION

METHOD M_CancelAction
VAR_INPUT
	eAction : E_Action;
END_VAR
CASE eAction OF
	E_Action.ACTION_SetPressure:
		IF bSetPress THEN
			fbSetPress(bExecute:= FALSE, pPneuChannelRef:= pPneuChannelPress);
		END_IF
	
	E_Action.ACTION_SetVacuum:
		IF bSetVacuum THEN
			fbSetVacuum(bExecute:= FALSE, pPneuChannelRef:= pPneuChannelVac);
		END_IF
		
	E_Action.ACTION_SwitchPressure:
		IF bSwitchPress AND nStateA_SwitchPress < 70 THEN
			nStateA_SwitchPress := 70;
		END_IF

	E_Action.ACTION_LockUnlock:
		IF bLockUnlock AND nStateA_LockUnlock < 70 THEN
			nStateA_LockUnlock := 70;
		END_IF	

	E_Action.ACTION_Expose:
		IF bExpose AND nStateA_Expose < 70 THEN
			nStateA_Expose := 70;
		END_IF

	E_Action.ACTION_PulsePressure:
		IF bPulsePress AND nStateA_PulsePress < 70 THEN
			nStateA_PulsePress := 70;
		END_IF	
ELSE
	SUPER^.M_CancelAction(eAction);
END_CASE
END_METHOD

PROPERTY P_stAbsPosPhys : ST_3DPoint
GET
VAR
	stTemp	: ST_3DPoint;
	stDim	: ST_3DDimension;
END_VAR
//Die absolute Postion eines Tool in "Z" hat nicht den gleichen Bezug wie X und Y
//X und Y beziehen sich auf den Koordinatenursprung, wenn die Achsen theoretischn aus Antrieb (0;0) stehen
//Z bezieht sich auf die Sliderunterkante des Z-Antriebes verechnet mit AbsPos vom Head(Ergebnis ist in den meisten Fällen negativ)

//Offset und RelPos addieren
stTemp := F_Add3DPoints(stRelPos,stOffset);

//in Abhängigkeit von LockState und Stempel aufgenommen die verschiedenen ZOffsets addieren
IF pFbMultiZ^.stStampSupport.bLocked THEN
	IF pFbMultiZ^.stStampSupport.bStampInSupport THEN
		//Offsets dem Stempeln verrechnen
		IF pPiece > 0 THEN
			stDim := pPiece^.P_stDimension;
			IF NOT pPiece^.P_bIgnoreOffset THEN
				stTemp := F_Add3DPoints(stTemp,pPiece^.P_stOffset);	
			END_IF
 			stTemp.Z := stTemp.Z + pPiece^.P_rZOverlapTool - stDim.Height;
		END_IF
	ELSE
		stTemp.Z := stTemp.Z + rZOffsetLocked;
	END_IF
ELSE //unlocked
	stTemp.Z := stTemp.Z + rZOffsetUnlocked;
END_IF

//AbsPos vom ParentSlot holen
IF pParentSlot > 0 THEN
	stTemp := F_Add3DPoints(stTemp,pParentSlot^.P_stAbsPos);	
END_IF
P_stAbsPosPhys := stTemp;
END_GET
END_PROPERTY

END_FUNCTION_BLOCK

// ---- Hardware/MultiZ/FB_MultiZStamp.TcPOU
FUNCTION_BLOCK FB_MultiZStamp
VAR_INPUT
END_VAR
VAR_OUTPUT
	bBusy : BOOL;
	bError : BOOL;
	nErrorId : ERRORID;
END_VAR
VAR
	bSendUnlockOffset : BOOL;
	bSendUnlockOffsetFlag : BOOL := TRUE;
	nUnlockOffset : DINT;
	
	bSwitchLight : BOOL;
	bSwitchLightFlag : BOOL := TRUE;
	bLight : BOOL;

	fbSdoWrite	: FB_SDO_WRITE;

	bInit : BOOL;
	bLockUnlock : BOOL;
	bAdjust : BOOL;
	
	tmrTimeout : TON;
	nCycleCounter : USINT;
	nStateAction : USINT;
	nStateActionNext : USINT;
	bActionFlag : BOOL := TRUE;
END_VAR

VAR_IN_OUT
	pFbMultiZ : POINTER TO FB_MultiZRef;
END_VAR

IF bSendUnlockOffset THEN
	IF bSendUnlockOffsetFlag XOR fbSdoWrite.bBusy THEN
		bSendUnlockOffsetFlag := FALSE;
		fbSdoWrite(sADSNetID:= pFbMultiZ^.P_sAdsNetId, nPortNr:= pFbMultiZ^.P_nAdsPort,
					nIndex:= cuCPUnlockOffset.nIndex, nSubIndex:= cuCPUnlockOffset.nSubIndex, 
					nDataLength:= cuCPUnlockOffset.nLength, nData:= pFbMultiZ^.stStampSupport.nUnlockOffset, bExecute:= TRUE);
	END_IF
	
	IF NOT fbSdoWrite.bBusy THEN
		IF fbSdoWrite.bError THEN
			bError := TRUE;
			nErrorId := fbSdoWrite.nAdsErrorId;
		ELSE
			nUnlockOffset := pFbMultiZ^.stStampSupport.nUnlockOffset;
		END_IF
		fbSdoWrite(bExecute:= FALSE);
		bSendUnlockOffsetFlag := TRUE;
		bSendUnlockOffset := FALSE;
	END_IF
END_IF

IF bSwitchLight THEN
	IF bSwitchLightFlag XOR fbSdoWrite.bBusy THEN
		bSwitchLightFlag := FALSE;
		fbSdoWrite(sADSNetID:= pFbMultiZ^.P_sAdsNetId, nPortNr:= pFbMultiZ^.P_nAdsPort,
					nIndex:= cuCPLight.nIndex, nSubIndex:= cuCPLight.nSubIndex, 
					nDataLength:= cuCPLight.nLength, nData:= BOOL_TO_DINT(pFbMultiZ^.stStampSupport.bLight), bExecute:= TRUE);
	END_IF
	
	IF NOT fbSdoWrite.bBusy THEN
		IF fbSdoWrite.bError THEN
			bError := TRUE;
			nErrorId := fbSdoWrite.nAdsErrorId;
		ELSE
			bLight := pFbMultiZ^.stStampSupport.bLight;
		END_IF
		fbSdoWrite(bExecute:= FALSE);
		bSwitchLightFlag := TRUE;
		bSwitchLight := FALSE;
	END_IF	
END_IF

IF bInit THEN
	A_Init();
	IF nStateAction >= 80 THEN
		IF nStateAction >= 99 THEN
			bError := TRUE;			
		END_IF
		nStateAction := 0;
		bInit := FALSE;
	END_IF
END_IF

IF bLockUnlock THEN
	A_LockUnlock();
	IF nStateAction >= 80 THEN
		IF nStateAction >= 99 THEN
			bError := TRUE;			
		END_IF
		nStateAction := 0;
		bLockUnlock := FALSE;
	END_IF	
END_IF

IF bAdjust THEN
	A_Adjust();
	IF nStateAction >= 80 THEN
		IF nStateAction >= 99 THEN
			bError := TRUE;			
		END_IF
		nStateAction := 0;
		bAdjust := FALSE;
	END_IF	
END_IF

IF NOT (bInit OR bLockUnlock OR bAdjust) THEN 
	bBusy := FALSE;
END_IF

PROPERTY P_nUnlockOffset : DINT
SET
IF pFbMultiZ > 0 THEN
	IF pFbMultiZ^.stStampSupport.nUnlockOffset <> P_nUnlockOffset THEN
		pFbMultiZ^.stStampSupport.nUnlockOffset := P_nUnlockOffset;
		bSendUnlockOffset := TRUE;
	END_IF
END_IF
END_SET
GET
IF pFbMultiZ > 0 THEN
	P_nUnlockOffset := nUnlockOffset;
END_IF
END_GET
END_PROPERTY

PROPERTY P_bStampInSupport : BOOL
GET
P_bStampInSupport := pFbMultiZ^.stStampSupport.bStampInSupport;
END_GET
END_PROPERTY

PROPERTY P_bLight : BOOL
GET
P_bLight := bLight;
END_GET
SET
IF pFbMultiZ > 0 THEN
	IF pFbMultiZ^.stStampSupport.bLight <> P_bLight THEN
		pFbMultiZ^.stStampSupport.bLight := P_bLight;
		bSwitchLight := TRUE;
	END_IF
END_IF
END_SET
END_PROPERTY

ACTION A_Adjust:
CASE nStateAction OF
	0:	//Mode auf "2" setzen
		IF bActionFlag XOR fbSdoWrite.bBusy THEN
			fbSdoWrite.nIndex := cuCPMode.nIndex;
			fbSdoWrite.nSubIndex := cuCPMode.nSubIndex;
			fbSdoWrite.nDataLength := cuCPMode.nLength;
			fbSdoWrite.nData := 2;			
			nStateAction := 50;
			nStateActionNext := 1;
		END_IF
		
	1:	//Ctrl auf "0" setzen
		IF bActionFlag XOR fbSdoWrite.bBusy THEN
			fbSdoWrite.nIndex := cuCPCtrl.nIndex;
			fbSdoWrite.nSubIndex := cuCPCtrl.nSubIndex;
			fbSdoWrite.nDataLength := cuCPCtrl.nLength;
			fbSdoWrite.nData := 0;			
			nStateAction := 50;
			nStateActionNext := 2;
		END_IF
		
	2:	//Winkel senden (Value wird in M_Adjust() geschrieben
		IF bActionFlag XOR fbSdoWrite.bBusy THEN
			fbSdoWrite.nIndex := cuCPAngleSetpoint.nIndex;
			fbSdoWrite.nSubIndex := cuCPAngleSetpoint.nSubIndex;
			fbSdoWrite.nDataLength := cuCPAngleSetpoint.nLength;
			fbSdoWrite.nData := INT_TO_DINT(pFbMultiZ^.stStampSupport.nAngleSetpoint);			
			nStateAction := 50;
			nStateActionNext := 3;
		END_IF
		
	3:	//Ctrl auf "1" setzen
		IF bActionFlag XOR fbSdoWrite.bBusy THEN
			fbSdoWrite.nIndex := cuCPCtrl.nIndex;
			fbSdoWrite.nSubIndex := cuCPCtrl.nSubIndex;
			fbSdoWrite.nDataLength := cuCPCtrl.nLength;
			fbSdoWrite.nData := 1;			
			nStateAction := 50;
			nStateActionNext := 4;
			nCycleCounter := 0;
		END_IF
		
	4:	nCycleCounter := nCycleCounter + 1;
		IF nCycleCounter = 5 THEN
			nStateAction := 5;
		END_IF

	5:	//Ctrl auf "0" setzen
		IF bActionFlag XOR fbSdoWrite.bBusy THEN
			fbSdoWrite.nIndex := cuCPCtrl.nIndex;
			fbSdoWrite.nSubIndex := cuCPCtrl.nSubIndex;
			fbSdoWrite.nDataLength := cuCPCtrl.nLength;
			fbSdoWrite.nData := 0;				
			nStateAction := 50;
			nStateActionNext := 6;
		END_IF		
		
 	6:	//Warten bis eingestellter Winkel erreicht
		tmrTimeout(IN:= TRUE, PT:=T#5S);
		IF pFbMultiZ^.stStampSupport.bAngleReached THEN
			tmrTimeout(IN:= FALSE);
			nStateAction := 80;
		END_IF
		
		IF tmrTimeout.Q THEN
			tmrTimeout(IN:= FALSE);
			bError := TRUE;
			nErrorId := E_ErrorIdCmd.ERRORID_TimeOut;
			nStateAction := 99;
		END_IF
END_CASE

IF nStateAction = 50 THEN
	IF bActionFlag XOR fbSdoWrite.bBusy THEN
		bActionFlag := FALSE;
		fbSdoWrite(sADSNetID:= pFbMultiZ^.P_sAdsNetId, nPortNr:= pFbMultiZ^.P_nAdsPort, bExecute:= TRUE);
	END_IF
	
	IF NOT fbSdoWrite.bBusy THEN
		IF fbSdoWrite.bError THEN
			bError := TRUE;
			nErrorId := fbSdoWrite.nAdsErrorId;
			nStateAction := 99;
		ELSE
			nStateAction := nStateActionNext;
		END_IF
		fbSdoWrite(bExecute:= FALSE);
		bActionFlag := TRUE;
	END_IF
END_IF

IF nStateAction = 70 THEN
	fbSdoWrite(bExecute:= FALSE);
	bActionFlag := TRUE;
	tmrTimeout(IN:= FALSE);
	nStateAction := 80;
END_IF
END_ACTION

ACTION A_LockUnlock:
CASE nStateAction OF
	0:	//Mode auf "1" setzen
		IF bActionFlag XOR fbSdoWrite.bBusy THEN
			//pFbMultiZ^.stStampSupport.nMode := 1;
			fbSdoWrite.nIndex := cuCPMode.nIndex;
			fbSdoWrite.nSubIndex := cuCPMode.nSubIndex;
			fbSdoWrite.nDataLength := cuCPMode.nLength;
			fbSdoWrite.nData := 1;
			nStateAction := 50;
			nStateActionNext := 1;
		END_IF
		
	1:	//Ctrl auf "0" setzen
		IF bActionFlag XOR fbSdoWrite.bBusy THEN
			//pFbMultiZ^.stStampSupport.bCtrl := 0;
			//fbSendSdoVar.eSdoVariType := E_MzSdoVariType.VARITYPE_uCPCtrl;
			fbSdoWrite.nIndex := cuCPCtrl.nIndex;
			fbSdoWrite.nSubIndex := cuCPCtrl.nSubIndex;
			fbSdoWrite.nDataLength := cuCPCtrl.nLength;
			fbSdoWrite.nData := 0;
			nStateAction := 50;
			nStateActionNext := 2;
		END_IF
		
	2:	//Lock senden (Value wird in M_LokcUnLock() geschrieben
		IF bActionFlag XOR fbSdoWrite.bBusy THEN
			//fbSendSdoVar.eSdoVariType := E_MzSdoVariType.VARITYPE_uCPLock;
			fbSdoWrite.nIndex := cuCPLock.nIndex;
			fbSdoWrite.nSubIndex := cuCPLock.nSubIndex;
			fbSdoWrite.nDataLength := cuCPLock.nLength;
			fbSdoWrite.nData := BOOL_TO_DINT(pFbMultiZ^.stStampSupport.bLock);
			nStateAction := 50;
			nStateActionNext := 3;
		END_IF
		
	3:	//Ctrl auf "1" setzen
		IF bActionFlag XOR fbSdoWrite.bBusy THEN
			//pFbMultiZ^.stStampSupport.bCtrl := 1;
			//fbSendSdoVar.eSdoVariType := E_MzSdoVariType.VARITYPE_uCPCtrl;
			fbSdoWrite.nIndex := cuCPCtrl.nIndex;
			fbSdoWrite.nSubIndex := cuCPCtrl.nSubIndex;
			fbSdoWrite.nDataLength := cuCPCtrl.nLength;
			fbSdoWrite.nData := 1;			
			nStateAction := 50;
			nStateActionNext := 4;
		END_IF		
		
	4:	//Timer (wozu das?)
		tmrTimeout(IN:= TRUE, PT:=T#1S);
		IF tmrTimeout.Q THEN
			tmrTimeout(IN:= FALSE);
			nStateAction := 5;
		END_IF
		
	5:	//Ctrl auf "0" setzen
		IF bActionFlag XOR fbSdoWrite.bBusy THEN
			//pFbMultiZ^.stStampSupport.bCtrl := 0;
			//fbSendSdoVar.eSdoVariType := E_MzSdoVariType.VARITYPE_uCPCtrl;
			fbSdoWrite.nIndex := cuCPCtrl.nIndex;
			fbSdoWrite.nSubIndex := cuCPCtrl.nSubIndex;
			fbSdoWrite.nDataLength := cuCPCtrl.nLength;
			fbSdoWrite.nData := 0;			
			nStateAction := 50;
			nStateActionNext := 6;
		END_IF

 	6:	//Warten, bis LockState erreicht
		tmrTimeout(IN:= TRUE, PT:=T#5S);
		IF pFbMultiZ^.stStampSupport.bLocked = pFbMultiZ^.stStampSupport.bLock THEN
			tmrTimeout(IN:= FALSE);
			nStateAction := 80;
		END_IF
		
		IF tmrTimeout.Q THEN
			tmrTimeout(IN:= FALSE);
			bError := TRUE;
			nErrorId := E_ErrorIdCmd.ERRORID_TimeOut;
			nStateAction := 99;
		END_IF
END_CASE

IF nStateAction = 50 THEN
	IF bActionFlag XOR fbSdoWrite.bBusy THEN
		bActionFlag := FALSE;
		fbSdoWrite(sADSNetID:= pFbMultiZ^.P_sAdsNetId, nPortNr:= pFbMultiZ^.P_nAdsPort, bExecute:= TRUE);
	END_IF
	
	IF NOT fbSdoWrite.bBusy THEN
		IF fbSdoWrite.bError THEN
			bError := TRUE;
			nErrorId := fbSdoWrite.nAdsErrorId;
			nStateAction := 99;
		ELSE
			nStateAction := nStateActionNext;
		END_IF
		fbSdoWrite(bExecute:= FALSE);
		bActionFlag := TRUE;
	END_IF
END_IF

IF nStateAction = 70 THEN
	tmrTimeout(IN:= FALSE);
	fbSdoWrite(bExecute:= FALSE);
	bActionFlag := TRUE;
	nStateAction := 80;
END_IF
END_ACTION

METHOD M_LockUnLock : ERRORID
VAR_INPUT
	bLock : BOOL;
END_VAR
IF pFbMultiZ^.stStampSupport.bLocked = bLock THEN
	RETURN;
ELSE
	IF NOT bBusy THEN
		pFbMultiZ^.stStampSupport.bLock := bLock;
		bBusy := TRUE;
		bLockUnlock := TRUE;
	END_IF
END_IF
END_METHOD

METHOD M_Adjust : ERRORID
VAR_INPUT
	nAngle : INT;
END_VAR
IF pFbMultiZ^.stStampSupport.nAngleSetpoint = nAngle THEN
	RETURN;
ELSE
	IF NOT bBusy THEN
		pFbMultiZ^.stStampSupport.nAngleSetpoint := nAngle;
		bBusy := TRUE;
		bAdjust := TRUE;
	END_IF
END_IF
END_METHOD

METHOD M_Init : ERRORID
VAR_INPUT
END_VAR
IF NOT bInit THEN
	bInit := TRUE;
	bBusy := TRUE;
END_IF
END_METHOD

ACTION A_Init:
CASE nStateAction OF
	0:	//Mode auf "6" setzen
		IF bActionFlag XOR fbSdoWrite.bBusy THEN
			fbSdoWrite.nIndex := cuCPMode.nIndex;
			fbSdoWrite.nSubIndex := cuCPMode.nSubIndex;
			fbSdoWrite.nDataLength := cuCPMode.nLength;
			fbSdoWrite.nData := 6; //OperationsMode
			nStateAction := 50;
			nStateActionNext := 1;
		END_IF	
		
	1:	//Ctrl auf "0" setzen
		IF bActionFlag XOR fbSdoWrite.bBusy THEN
			fbSdoWrite.nIndex := cuCPCtrl.nIndex;
			fbSdoWrite.nSubIndex := cuCPCtrl.nSubIndex;
			fbSdoWrite.nDataLength := cuCPCtrl.nLength;
			fbSdoWrite.nData := 0;
			nStateAction := 50;
			nStateActionNext := 2;
		END_IF		
		
	2:	//Ctrl auf "1" setzen
		IF bActionFlag XOR fbSdoWrite.bBusy THEN
			fbSdoWrite.nIndex := cuCPCtrl.nIndex;
			fbSdoWrite.nSubIndex := cuCPCtrl.nSubIndex;
			fbSdoWrite.nDataLength := cuCPCtrl.nLength;
			fbSdoWrite.nData := 1;
			nStateAction := 50;
			nStateActionNext := 3;
		END_IF			
		
	3:	//Angle auf "0" setzen
		IF bActionFlag XOR fbSdoWrite.bBusy THEN
			fbSdoWrite.nIndex := cuCPAngleSetpoint.nIndex;
			fbSdoWrite.nSubIndex := cuCPAngleSetpoint.nSubIndex;
			fbSdoWrite.nDataLength := cuCPAngleSetpoint.nLength;
			fbSdoWrite.nData := 0;			
			nStateAction := 50;
			nStateActionNext := 4;
		END_IF	
		
	4:	//Warten bis Init ready
		tmrTimeout(IN:= TRUE, PT:=T#10S);
		IF tmrTimeout.Q THEN
			nStateAction := 99;
			nErrorId := E_ErrorIdCmd.ERRORID_TimeOut;
			tmrTimeout(IN:= FALSE);
		END_IF
		IF pFbMultiZ^.stStampSupport.bInitLockOk AND pFbMultiZ^.stStampSupport.bInitSpinOk THEN
			tmrTimeout(IN:= FALSE);
			nStateAction := 80;
		END_IF

END_CASE

IF nStateAction = 50 THEN
	IF bActionFlag XOR fbSdoWrite.bBusy THEN
		bActionFlag := FALSE;
		fbSdoWrite(sADSNetID:= pFbMultiZ^.P_sAdsNetId, nPortNr:= pFbMultiZ^.P_nAdsPort, bExecute:= TRUE);
	END_IF
	
	IF NOT fbSdoWrite.bBusy THEN
		IF fbSdoWrite.bError THEN
			bError := TRUE;
			nErrorId := fbSdoWrite.nAdsErrorId;
			nStateAction := 99;
		ELSE
			nStateAction := nStateActionNext;
		END_IF
		fbSdoWrite(bExecute:= FALSE);
		bActionFlag := TRUE;
	END_IF
END_IF

IF nStateAction = 70 THEN
	tmrTimeout(IN:= FALSE);
	fbSdoWrite(bExecute:= FALSE);
	bActionFlag := TRUE;
	nStateAction := 80;
END_IF
END_ACTION

METHOD M_Reset
VAR_INPUT
END_VAR
bError := FALSE;
nErrorId := 0;
END_METHOD

METHOD M_Stop
VAR_INPUT
END_VAR
IF bBusy THEN
	nStateAction := 70;
END_IF
END_METHOD

PROPERTY P_bStampInMagazine : BOOL
GET
P_bStampInMagazine := pFbMultiZ^.stStampSupport.bStampInMagazine;
END_GET
END_PROPERTY

END_FUNCTION_BLOCK

// ---- Objects/Targets/Passive/FB_StampMagazine.TcPOU
FUNCTION_BLOCK FB_StampMagazine EXTENDS FB_Rack IMPLEMENTS I_TargetZSensor
VAR
	//Spec-Properties
	nNoOfSpecPoints	: USINT;
	stMeasurePoint	: ST_3DPoint;
	stOffsetStampDetect : ST_3DPoint;
	
	bSensor AT %I* : BOOL;
END_VAR

METHOD FB_init : BOOL
VAR_INPUT
	bInitRetains : BOOL; // if TRUE, the retain variables are initialized (warm start / cold start)
	bInCopyCode : BOOL;  // if TRUE, the instance afterwards gets moved into the copy code (online change)
END_VAR
eObjectType := E_ObjectType.OBJECTTYPE_StampMagazine;
eObjectGroup := E_ObjectGroup.OBJECTGROUP_Target OR E_ObjectGroup.OBJECTGROUP_Rack;
END_METHOD

METHOD M_AddChild : ERRORID
VAR_INPUT
	pObject : POINTER TO FB_Object;
	nSlotNr	: UINT;
	nIndex 	: INT;
END_VAR
//Kann folgende Objekte aufnehmen:
IF pObject > 0 THEN
	IF pObject^.P_eObjectType = E_ObjectType.OBJECTTYPE_Point THEN
		M_AddChild := SUPER^.M_AddChild(pObject,nSlotNr,nIndex);
	ELSIF pObject^.P_eObjectType = E_ObjectType.OBJECTTYPE_Stamp THEN
		//darf nur in ein Slot
		IF nSlotNr > 0 THEN
			M_AddChild := SUPER^.M_AddChild(pObject,nSlotNr,nIndex);
		ELSE
			M_AddChild := E_ErrorIdObjMgmt.ERRORID_InvalidSlotNumber;	
		END_IF
	ELSE
		M_AddChild := E_ErrorIdObjMgmt.ERRORID_InvalidParentObject;
	END_IF
ELSE
	M_AddChild := E_ErrorIdObjMgmt.ERRORID_InvalidParentObject;
END_IF
END_METHOD

METHOD M_CheckAction : ERRORID
VAR_INPUT
	refActionData 	: REFERENCE TO ST_ActionData;
	pCorrelObject	: POINTER TO FB_Object;
END_VAR

VAR
	pSlot : POINTER TO FB_PieceSlot;
END_VAR
IF refActionData.eAction = E_Action.ACTION_ExchangePiece THEN
	pSlot := super^.M_GetSlot(DINT_TO_UINT(refActionData.aParams[1]));
	IF pSlot = 0 THEN
		M_CheckAction := E_ErrorIdCmd.ERRORID_InvalidTargetSlot;
	ELSE
		IF refActionData.aParams[2] = 0 THEN //Drop - es darf kein Stamp im Slot sein
			IF pSlot^.P_pPiece > 0 THEN
				M_CheckAction := E_ErrorIdCmd.ERRORID_PieceAlreadyInSlot;	
			END_IF
		ELSIF refActionData.aParams[2] = 1 THEN //Take - es muss ein Stemple im Slot
			IF pSlot^.P_pPiece = 0 THEN
				M_CheckAction := E_ErrorIdCmd.ERRORID_NoPieceInSlot;	
			END_IF
		ELSE
			M_CheckAction := E_ErrorIdCmd.ERRORID_InvalidCtrl;		
		END_IF		
	END_IF
ELSE
	M_CheckAction := SUPER^.M_CheckAction(refActionData, pCorrelObject);
END_IF
END_METHOD

METHOD M_ClearAllProps
VAR_INPUT
	bIgnoreParent : BOOL; //Es wird das gesamte OD gelöscht. -> Zeiger auf Parent nicht mehr gültig!
END_VAR
SUPER^.M_ClearAllProps(bIgnoreParent);
END_METHOD

METHOD M_GetAbsPos : ST_3DPoint
VAR_INPUT
	pChildPos	: POINTER TO ST_3DPoint;
	eTargetRef 	: E_TargetRef;
	nParam1		: UINT;
 	nParam2		: UINT;
	nParam3		: USINT;
	nParam4		: USINT;
	nZLevel		: USINT;
END_VAR
VAR_OUTPUT
	nErrorId 	: ERRORID;
	lrAngle		: LREAL;
END_VAR
VAR
	stLocPosLB : ST_3DPoint;
END_VAR
IF eTargetRef = E_TargetRef.TARGETREF_SpecPoint THEN
	IF nParam1 = 1 AND nNoOfSpecPoints = 1 THEN	//MeasurePoint
		stLocPosLB := P_stRelPosLB; //linke untere Ecke StampMagazine
		stLocPosLB := F_Add3DPoints(stLocPosLB,stMeasurePoint);
	
		M_GetAbsPos := pParentTarget^.M_GetAbsPos(pChildPos := ADR(stLocPosLB), eTargetRef:= E_TargetRef.TARGETREF_LeftBottom,
													nParam1:= 0,
													nParam2:= 0, nParam3:= 0, nParam4:= 0, nZLevel:= 0,
													lrAngle => lrAngle, nErrorId=> nErrorId);
	ELSE
		nErrorId := E_ErrorIdCmd.ERRORID_InvalidTargetPointNr;
	END_IF	
ELSE
	M_GetAbsPos := SUPER^.M_GetAbsPos(pChildPos := pChildPos, eTargetRef:= eTargetRef,
													nParam1:= nParam1,
													nParam2:= nParam2, nParam3:= nParam3, nParam4:= 0, nZLevel:= nZLevel,
													lrAngle => lrAngle, nErrorId=> nErrorId);
END_IF
END_METHOD

METHOD M_GetAllProps : ERRORID
VAR_INPUT
	refCmdData : REFERENCE TO  ST_CmdData;
END_VAR

VAR
	i : USINT;
END_VAR
SUPER^.M_GetAllProps(refCmdData);

//MeasurePoint
nCurrentPropIndex := nCurrentPropIndex + 1;
refCmdData.n32Data[nCurrentPropIndex] := nNoOfSpecPoints;
FOR i:= 1 TO nNoOfSpecPoints BY 1 DO
	nCurrentPropIndex := nCurrentPropIndex + 1;
	refCmdData.n32Data[nCurrentPropIndex] := REAL_TO_DINT(stMeasurePoint.X);
	nCurrentPropIndex := nCurrentPropIndex + 1;
	refCmdData.n32Data[nCurrentPropIndex] := REAL_TO_DINT(stMeasurePoint.Y);
	nCurrentPropIndex := nCurrentPropIndex + 1;
	refCmdData.n32Data[nCurrentPropIndex] := REAL_TO_DINT(stMeasurePoint.Z);	
END_FOR

nCurrentPropIndex := nCurrentPropIndex + 1; 
refCmdData.n32Data[nCurrentPropIndex] := REAL_TO_DINT(stOffsetStampDetect.X);
nCurrentPropIndex := nCurrentPropIndex + 1; 
refCmdData.n32Data[nCurrentPropIndex] := REAL_TO_DINT(stOffsetStampDetect.Y);
nCurrentPropIndex := nCurrentPropIndex + 1; 
refCmdData.n32Data[nCurrentPropIndex] := REAL_TO_DINT(stOffsetStampDetect.Z);
END_METHOD

METHOD M_SetAllProps : ERRORID
VAR_INPUT
	refCmdData : REFERENCE TO  ST_CmdData;
END_VAR

VAR
END_VAR
M_SetAllProps := SUPER^.M_SetAllProps(refCmdData);

IF M_SetAllProps > 0 THEN
	RETURN;
END_IF

//MeasurePoint
nCurrentPropIndex := nCurrentPropIndex + 1;
nSpecPropIndex := nCurrentPropIndex;
nNoOfSpecPoints := DINT_TO_USINT(refCmdData.n32Data[nCurrentPropIndex]);
IF nNoOfSpecPoints = 0 THEN
	;
ELSIF nNoOfSpecPoints = 1 THEN
	nCurrentPropIndex := nCurrentPropIndex + 1;
	stMeasurePoint.X := DINT_TO_REAL(refCmdData.n32Data[nCurrentPropIndex]);
	nCurrentPropIndex := nCurrentPropIndex + 1;
	stMeasurePoint.Y := DINT_TO_REAL(refCmdData.n32Data[nCurrentPropIndex]);
	nCurrentPropIndex := nCurrentPropIndex + 1;
	stMeasurePoint.Z := DINT_TO_REAL(refCmdData.n32Data[nCurrentPropIndex]);	
ELSE
	M_SetAllProps := E_ErrorIdObjMgmt.ERRORID_InvalidNoOfSpecPoints;
END_IF

nCurrentPropIndex := nCurrentPropIndex + 1;
stOffsetStampDetect.X := DINT_TO_REAL(refCmdData.n32Data[nCurrentPropIndex]);
nCurrentPropIndex := nCurrentPropIndex + 1;
stOffsetStampDetect.Y := DINT_TO_REAL(refCmdData.n32Data[nCurrentPropIndex]);
nCurrentPropIndex := nCurrentPropIndex + 1;
stOffsetStampDetect.Z := DINT_TO_REAL(refCmdData.n32Data[nCurrentPropIndex]);

nNoOfProps := nCurrentPropIndex + 1;
END_METHOD

METHOD M_SetSingleProp : ERRORID
VAR_INPUT
	refCmdData : REFERENCE TO  ST_CmdData;
END_VAR
IF nSpecPropIndex = refCmdData.aHeader[1] THEN
	stMeasurePoint.X := DINT_TO_REAL(refCmdData.n32Data[0]);
ELSIF (nSpecPropIndex + 1) = refCmdData.aHeader[1] THEN
	stMeasurePoint.Y := DINT_TO_REAL(refCmdData.n32Data[0]);
ELSIF (nSpecPropIndex + 2) = refCmdData.aHeader[1] THEN
	stMeasurePoint.Z := DINT_TO_REAL(refCmdData.n32Data[0]);
ELSIF (nSpecPropIndex + 3) = refCmdData.aHeader[1] THEN
	stOffsetStampDetect.X := DINT_TO_REAL(refCmdData.n32Data[0]);
ELSIF (nSpecPropIndex + 4) = refCmdData.aHeader[1] THEN
	stOffsetStampDetect.Y := DINT_TO_REAL(refCmdData.n32Data[0]);
ELSIF (nSpecPropIndex + 5) = refCmdData.aHeader[1] THEN
	stOffsetStampDetect.Z := DINT_TO_REAL(refCmdData.n32Data[0]);
ELSE
	M_SetSingleProp := SUPER^.M_SetSingleProp(refCmdData);
END_IF
END_METHOD

PROPERTY P_bMeasurePointAvailable : BOOL
GET
IF nNoOfSpecPoints > 0 THEN
	P_bMeasurePointAvailable := TRUE;
END_IF
END_GET
END_PROPERTY

PROPERTY P_bSensor : BOOL
GET
P_bSensor := NOT bSensor;
END_GET
END_PROPERTY

PROPERTY P_stOffsetStampDetect : ST_3DPoint
GET
P_stOffsetStampDetect := stOffsetStampDetect;
END_GET
SET
stOffsetStampDetect := P_stOffsetStampDetect;
END_SET
END_PROPERTY

END_FUNCTION_BLOCK

// ---- Objects/Tools/FB_DeloDot.TcPOU
FUNCTION_BLOCK FB_DeloDot EXTENDS FB_GCodeTool
VAR_INPUT
END_VAR
VAR_OUTPUT
END_VAR
VAR
	//Reference zu TripleTrigger
	pTripleTrigRef 		: POINTER TO FB_HwRefTripleTrigger;
	pPneuChannelPress	: POINTER TO FB_PneuChannelRef;
	
	//Specproperties
	nSubType			: DINT;		//wird noch nicht ausgewertet
	nTriggerChannel		: USINT;
	nStroke				: UINT;
	
	nDOutChanValvePress	: USINT;	//Digitaler Ausgangskanal MzHead Druckventil
	
	//****************************************Aktionvariablen****************************************************
	
	stActionDataSpec	: ST_ActionData;
	
	//Action: "SetPressure"
	bSetPress			: BOOL;
	fbSetPress			: FB_SetPressure;
	
	//Action: "SwitchPressure"
	bSwitchPress		: BOOL;			
	nStateA_SwitchPress	: USINT;		//State von A_SwitchPress()
	nPressValue			: INT;			//Solldruck
	//bPressOn			: BOOL;			//Druckventil "Auf"
	eSwitchPressCtrl	: E_PressCtrl;
	tPressTime			: TIME;			//nach dieser Zeit Ventil automatisch wieder zu
	timerPress			: TON;			//Timer für Öffnungszeit Druckventil 	
	
	//Action: "InitTool"
	bInitTool			: BOOL;
	nStateA_InitTool	: USINT;
	
	//Action: "Dispense"
	bDispense				: BOOL;
	nStateA_Dispense		: USINT;
	nDrops					: UINT;
	bDispenseStart			: BOOL;
	
END_VAR

IF eCurrentState = E_MachineState.MACHINESTATE_Active THEN
	IF bInitTool THEN
		A_InitTool();
		IF nStateA_InitTool >= 80 THEN
			IF nStateA_InitTool >= 99 THEN
				bError := TRUE;
			END_IF
			bInitTool := FALSE;
			nStateA_InitTool := 0;
			M_RemoveListEntry(nSearchValue:= E_Action.ACTION_Init);
		END_IF		
	END_IF

	IF bSetPress THEN
		fbSetPress(pPneuChannelRef:= pPneuChannelPress);
		IF NOT fbSetPress.bBusy THEN
			IF fbSetPress.bError THEN
				bError := TRUE;
				stError.ErrorId := fbSetPress.nErrorId;
				stError.POU := E_POU.POU_FB_Luer;
				fbErrorList.M_Add(stError);
			END_IF
			bSetPress := FALSE;
			fbSetPress(pPneuChannelRef:= pPneuChannelPress, bExecute:= FALSE);
			M_RemoveListEntry(nSearchValue:= E_Action.ACTION_SetPressure);
		END_IF
	END_IF	
	
	IF bSwitchPress THEN	//Kartuschendruck einstellen und Ein-bzw. Aus schalten 
		A_SwitchPress();
		IF nStateA_SwitchPress >= 80 THEN
			IF nStateA_SwitchPress >= 99 THEN
				bError := TRUE;	
			END_IF
			bSwitchPress := FALSE;
			nStateA_SwitchPress := 0;
			M_RemoveListEntry(nSearchValue:= E_Action.ACTION_SwitchPressure);
		END_IF
	END_IF

	IF bDispense THEN
		A_Dispense();
		IF nStateA_Dispense >= 80 THEN
			IF nStateA_Dispense >= 99 THEN
				bError := TRUE;	
			END_IF
			bDispense := FALSE;
			nStateA_Dispense := 0;
			M_RemoveListEntry(nSearchValue:= E_Action.ACTION_DispenseDrops);
		END_IF
	END_IF
END_IF

SUPER^();	//FB_MzTool aufrufen

//Prozessdaten aktualisieren
IF pPneuChannelPress > 0 THEN
	stProcessData.n32Data[7] := pPneuChannelPress^.P_nCurrentPressure;
END_IF

IF pFbMultiZ > 0 THEN
	IF nDOutChanValvePress > 0 AND nDOutChanValvePress < 8 THEN
		stProcessData.n32Data[8] := BOOL_TO_DINT(pFbMultiZ^.aDigiOut[nDOutChanValvePress]);
	END_IF
END_IF

IF pTripleTrigRef > 0 THEN
	stProcessData.n32Data[9] := BOOL_TO_DINT(pTripleTrigRef^.M_GetState(nTriggerChannel));
END_IF

aObjProcData[nNotifyId] := stProcessData;

ACTION A_Dispense:
CASE nStateA_Dispense OF
	0:
		pTripleTrigRef^.M_TriggerOn(nTriggerChannel,nDrops);
		nStateA_Dispense := 1;

	1:	//Einen Zyklus warten
		nStateA_Dispense := 2;
		
	2:	//Warten bis Dispensen fertig
		IF NOT pTripleTrigRef^.M_GetState(nTriggerChannel) THEN
			pTripleTrigRef^.M_TriggerOff(nTriggerChannel);
			nStateA_Dispense := 80;
		END_IF
		
	70:	//Abbrechen
		pTripleTrigRef^.M_TriggerOff(nTriggerChannel);
		nStateA_Dispense := 80;
END_CASE
END_ACTION

ACTION A_InitTool:
nStateA_InitTool := 80;
END_ACTION

ACTION A_Reset:
//Ist noch eine Aktion aktiv?
IF nStateA_ResetSpec = 0 THEN
	IF bDispense THEN
		bDispense := FALSE;
		nStateA_Dispense := 0;
	END_IF
	
	IF bSetPress THEN
		bSetPress := FALSE;
		fbSetPress(bExecute:= FALSE, pPneuChannelRef:= pPneuChannelPress);
	END_IF
	
	IF bSwitchPress THEN
		bSwitchPress := FALSE;
		nStateA_SwitchPress := 0;
	END_IF
 
	nStateA_ResetSpec := 80;
END_IF

SUPER^.A_Reset();
END_ACTION

ACTION A_Stop:
IF nStateA_Stop = 0 THEN
	
	IF bSetPress THEN
		fbSetPress(bExecute:= FALSE, pPneuChannelRef:= pPneuChannelPress);
	END_IF

	IF bSwitchPress AND nStateA_SwitchPress < 70 THEN
		nStateA_SwitchPress := 70;
	END_IF
	
	IF bDispense AND nStateA_Dispense < 70 THEN
		nStateA_Dispense := 70;
	END_IF
	
	nStateA_Stop := 1;	
END_IF

SUPER^.A_Stop();
END_ACTION

ACTION A_SwitchPress:
CASE nStateA_SwitchPress OF
	0:	//Ventil Einschalten
		pFbMultiZ^.aDigiOut[nDOutChanValvePress] := TRUE;
	
		//Timer starten
		IF tPressTime = T#0S THEN
			nStateA_SwitchPress := 80;
			RETURN;	
		END_IF
		
		timerPress(IN:= TRUE, PT:= tPressTime);
		nStateA_SwitchPress := 1;
		
	1:	//Warten bis Zeitabgelaufen
		timerPress();
		IF timerPress.Q THEN
			timerPress(IN:= FALSE);
			pFbMultiZ^.aDigiOut[nDOutChanValvePress] := FALSE;
			nStateA_SwitchPress := 80;
		END_IF
		
	70:	//Abbrechen
		timerPress(IN:= FALSE);
		pFbMultiZ^.aDigiOut[nDOutChanValvePress] := FALSE;
		nStateA_SwitchPress := 80;
END_CASE
END_ACTION

METHOD FB_init : BOOL
VAR_INPUT
	bInitRetains : BOOL; // if TRUE, the retain variables are initialized (warm start / cold start)
	bInCopyCode : BOOL;  // if TRUE, the instance afterwards gets moved into the copy code (online change)
END_VAR
eObjectType := E_ObjectType.OBJECTTYPE_DeloDot;
eObjectGroup := E_ObjectGroup.OBJECTGROUP_MzTool OR E_ObjectGroup.OBJECTGROUP_Device;
END_METHOD

